gfCNCPoint3[27581] = {X 474.4193, Y 40.3571, Z -4.6667, A 0.000, B 0.000, C 0.000 }
gfCNCPoint3[27582] = {X 478.5504, Y 32.2710, Z -4.6667, A 0.000, B 0.000, C 0.000 }
gfCNCPoint3[27583] = {X 477.2666, Y 31.4237, Z -4.6667, A 0.000, B 0.000, C 0.000 }
gfCNCPoint3[27584] = {X 476.1107, Y 30.4089, Z -4.6667, A 0.000, B 0.000, C 0.000 }
gfCNCPoint3[27585] = {X 475.1043, Y 29.2457, Z -4.6667, A 0.000, B 0.000, C 0.000 }
gfCNCPoint3[27586] = {X 474.2663, Y 27.9559, Z -4.6667, A 0.000, B 0.000, C 0.000 }
gfCNCPoint3[27587] = {X 473.6124, Y 26.5637, Z -4.6667, A 0.000, B 0.000, C 0.000 }
gfCNCPoint3[27588] = {X 473.1548, Y 25.0952, Z -4.6667, A 0.000, B 0.000, C 0.000 }
gfCNCPoint3[27589] = {X 472.8451, Y 23.4362, Z -4.6667, A 0.000, B 0.000, C 0.000 }
gfCNCPoint3[27590] = {X 472.7065, Y 21.7542, Z -4.6667, A 0.000, B 0.000, C 0.000 }
gfCNCPoint3[27591] = {X 472.7407, Y 20.0669, Z -4.6667, A 0.000, B 0.000, C 0.000 }
gfCNCPoint3[27592] = {X 472.9473, Y 18.3920, Z -4.6667, A 0.000, B 0.000, C 0.000 }
gfCNCPoint3[27593] = {X 473.3241, Y 16.7469, Z -4.6667, A 0.000, B 0.000, C 0.000 }
gfCNCPoint3[27594] = {X 473.8558, Y 15.2628, Z -4.6667, A 0.000, B 0.000, C 0.000 }
gfCNCPoint3[27595] = {X 474.5840, Y 13.8645, Z -4.6667, A 0.000, B 0.000, C 0.000 }
gfCNCPoint3[27596] = {X 475.4953, Y 12.5780, Z -4.6667, A 0.000, B 0.000, C 0.000 }
gfCNCPoint3[27597] = {X 476.5726, Y 11.4271, Z -4.6667, A 0.000, B 0.000, C 0.000 }
gfCNCPoint3[27598] = {X 477.7962, Y 10.4330, Z -4.6667, A 0.000, B 0.000, C 0.000 }
gfCNCPoint3[27599] = {X 479.1434, Y 9.6141, Z -4.6667, A 0.000, B 0.000, C 0.000 }
gfCNCPoint3[27600] = {X 480.5892, Y 8.9856, Z -4.6667, A 0.000, B 0.000, C 0.000 }
gfCNCPoint3[27601] = {X 482.1069, Y 8.5592, Z -4.6667, A 0.000, B 0.000, C 0.000 }
gfCNCPoint3[27602] = {X 484.1811, Y 8.2359, Z -4.6667, A 0.000, B 0.000, C 0.000 }
gfCNCPoint3[27603] = {X 486.2773, Y 8.1227, Z -4.6667, A 0.000, B 0.000, C 0.000 }
gfCNCPoint3[27604] = {X 486.9700, Y 8.1106, Z -4.6667, A 0.000, B 0.000, C 0.000 }
gfCNCPoint3[27605] = {X 492.3835, Y 8.1106, Z -4.6667, A 0.000, B 0.000, C 0.000 }
gfCNCPoint3[27606] = {X 492.3835, Y 4.1106, Z -4.6667, A 0.000, B 0.000, C 0.000 }
gfCNCPoint3[27607] = {X 492.3835, Y 8.1906, Z -4.6667, A 0.000, B 0.000, C 0.000 }
gfCNCPoint3[27608] = {X 502.2053, Y 8.1906, Z -4.6667, A 0.000, B 0.000, C 0.000 }
gfCNCPoint3[27609] = {X 502.7369, Y 8.1947, Z -4.6667, A 0.000, B 0.000, C 0.000 }
gfCNCPoint3[27610] = {X 503.6180, Y 8.3005, Z -4.6667, A 0.000, B 0.000, C 0.000 }
gfCNCPoint3[27611] = {X 504.4538, Y 8.5987, Z -4.6667, A 0.000, B 0.000, C 0.000 }
gfCNCPoint3[27612] = {X 505.2029, Y 9.0746, Z -4.6667, A 0.000, B 0.000, C 0.000 }
gfCNCPoint3[27613] = {X 505.8279, Y 9.7045, Z -4.6667, A 0.000, B 0.000, C 0.000 }
gfCNCPoint3[27614] = {X 506.2979, Y 10.4573, Z -4.6667, A 0.000, B 0.000, C 0.000 }
gfCNCPoint3[27615] = {X 506.5896, Y 11.2954, Z -4.6667, A 0.000, B 0.000, C 0.000 }
gfCNCPoint3[27616] = {X 506.6885, Y 12.1773, Z -4.6667, A 0.000, B 0.000, C 0.000 }
gfCNCPoint3[27617] = {X 506.6883, Y 13.0192, Z -4.6667, A 0.000, B 0.000, C 0.000 }
gfCNCPoint3[27618] = {X 506.5797, Y 13.9048, Z -4.6667, A 0.000, B 0.000, C 0.000 }
gfCNCPoint3[27619] = {X 506.2774, Y 14.7443, Z -4.6667, A 0.000, B 0.000, C 0.000 }
gfCNCPoint3[27620] = {X 505.7966, Y 15.4959, Z -4.6667, A 0.000, B 0.000, C 0.000 }
gfCNCPoint3[27621] = {X 505.1612, Y 16.1222, Z -4.6667, A 0.000, B 0.000, C 0.000 }
gfCNCPoint3[27622] = {X 505.1611, Y 41.0655, Z -4.6667, A 0.000, B 0.000, C 0.000 }
gfCNCPoint3[27623] = {X 505.3000, Y 41.1789, Z -4.6667, A 0.000, B 0.000, C 0.000 }
gfCNCPoint3[27624] = {X 505.8859, Y 41.8054, Z -4.6667, A 0.000, B 0.000, C 0.000 }
gfCNCPoint3[27625] = {X 506.3249, Y 42.5424, Z -4.6667, A 0.000, B 0.000, C 0.000 }
gfCNCPoint3[27626] = {X 506.5965, Y 43.3560, Z -4.6667, A 0.000, B 0.000, C 0.000 }
gfCNCPoint3[27627] = {X 506.6885, Y 44.2089, Z -4.6667, A 0.000, B 0.000, C 0.000 }
gfCNCPoint3[27628] = {X 506.6885, Y 45.0000, Z -4.6667, A 0.000, B 0.000, C 0.000 }
gfCNCPoint3[27629] = {X 506.5882, Y 45.8901, Z -4.6667, A 0.000, B 0.000, C 0.000 }
gfCNCPoint3[27630] = {X 506.2924, Y 46.7355, Z -4.6667, A 0.000, B 0.000, C 0.000 }
gfCNCPoint3[27631] = {X 505.8158, Y 47.4940, Z -4.6667, A 0.000, B 0.000, C 0.000 }
gfCNCPoint3[27632] = {X 505.1825, Y 48.1273, Z -4.6667, A 0.000, B 0.000, C 0.000 }
gfCNCPoint3[27633] = {X 504.4240, Y 48.6039, Z -4.6667, A 0.000, B 0.000, C 0.000 }
gfCNCPoint3[27634] = {X 503.5786, Y 48.8997, Z -4.6667, A 0.000, B 0.000, C 0.000 }
gfCNCPoint3[27635] = {X 502.6885, Y 49.0000, Z -4.6667, A 0.000, B 0.000, C 0.000 }
gfCNCPoint3[27636] = {X 496.2450, Y 49.0000, Z -4.6667, A 0.000, B 0.000, C 0.000 }
gfCNCPoint3[27637] = {X 495.3549, Y 48.8997, Z -4.6667, A 0.000, B 0.000, C 0.000 }
gfCNCPoint3[27638] = {X 494.5095, Y 48.6039, Z -4.6667, A 0.000, B 0.000, C 0.000 }
gfCNCPoint3[27639] = {X 493.7511, Y 48.1273, Z -4.6667, A 0.000, B 0.000, C 0.000 }
gfCNCPoint3[27640] = {X 493.1177, Y 47.4939, Z -4.6667, A 0.000, B 0.000, C 0.000 }
gfCNCPoint3[27641] = {X 492.6411, Y 46.7355, Z -4.6667, A 0.000, B 0.000, C 0.000 }
gfCNCPoint3[27642] = {X 492.3453, Y 45.8901, Z -4.6667, A 0.000, B 0.000, C 0.000 }
gfCNCPoint3[27643] = {X 492.2450, Y 45.0000, Z -4.6667, A 0.000, B 0.000, C 0.000 }
gfCNCPoint3[27644] = {X 492.2454, Y 44.1538, Z -4.6667, A 0.000, B 0.000, C 0.000 }
gfCNCPoint3[27645] = {X 492.3560, Y 43.2730, Z -4.6667, A 0.000, B 0.000, C 0.000 }
gfCNCPoint3[27646] = {X 492.6582, Y 42.4382, Z -4.6667, A 0.000, B 0.000, C 0.000 }
gfCNCPoint3[27647] = {X 493.1371, Y 41.6907, Z -4.6667, A 0.000, B 0.000, C 0.000 }
gfCNCPoint3[27648] = {X 493.7690, Y 41.0672, Z -4.6667, A 0.000, B 0.000, C 0.000 }
gfCNCPoint3[27649] = {X 493.7690, Y 34.1538, Z -4.6667, A 0.000, B 0.000, C 0.000 }
gfCNCPoint3[27650] = {X 490.7733, Y 34.1538, Z -4.6667, A 0.000, B 0.000, C 0.000 }
gfCNCPoint3[27651] = {X 490.5302, Y 34.1516, Z -4.6667, A 0.000, B 0.000, C 0.000 }
gfCNCPoint3[27652] = {X 486.0908, Y 42.7966, Z -4.6667, A 0.000, B 0.000, C 0.000 }
gfCNCPoint3[27653] = {X 486.1474, Y 42.9488, Z -4.6667, A 0.000, B 0.000, C 0.000 }
gfCNCPoint3[27654] = {X 486.2998, Y 43.5707, Z -4.6667, A 0.000, B 0.000, C 0.000 }
gfCNCPoint3[27655] = {X 486.3510, Y 44.2089, Z -4.6667, A 0.000, B 0.000, C 0.000 }
gfCNCPoint3[27656] = {X 486.3510, Y 45.0000, Z -4.6667, A 0.000, B 0.000, C 0.000 }
gfCNCPoint3[27657] = {X 486.2507, Y 45.8901, Z -4.6667, A 0.000, B 0.000, C 0.000 }
gfCNCPoint3[27658] = {X 485.9549, Y 46.7355, Z -4.6667, A 0.000, B 0.000, C 0.000 }
gfCNCPoint3[27659] = {X 485.4783, Y 47.4940, Z -4.6667, A 0.000, B 0.000, C 0.000 }
gfCNCPoint3[27660] = {X 484.8450, Y 48.1273, Z -4.6667, A 0.000, B 0.000, C 0.000 }
gfCNCPoint3[27661] = {X 484.0866, Y 48.6039, Z -4.6667, A 0.000, B 0.000, C 0.000 }
gfCNCPoint3[27662] = {X 483.2411, Y 48.8997, Z -4.6667, A 0.000, B 0.000, C 0.000 }
gfCNCPoint3[27663] = {X 482.3510, Y 49.0000, Z -4.6667, A 0.000, B 0.000, C 0.000 }
gfCNCPoint3[27664] = {X 475.7650, Y 49.0000, Z -4.6667, A 0.000, B 0.000, C 0.000 }
gfCNCPoint3[27665] = {X 474.8749, Y 48.8997, Z -4.6667, A 0.000, B 0.000, C 0.000 }
gfCNCPoint3[27666] = {X 474.0294, Y 48.6039, Z -4.6667, A 0.000, B 0.000, C 0.000 }
gfCNCPoint3[27667] = {X 473.2710, Y 48.1273, Z -4.6667, A 0.000, B 0.000, C 0.000 }
gfCNCPoint3[27668] = {X 472.6376, Y 47.4940, Z -4.6667, A 0.000, B 0.000, C 0.000 }
gfCNCPoint3[27669] = {X 472.1611, Y 46.7355, Z -4.6667, A 0.000, B 0.000, C 0.000 }
gfCNCPoint3[27670] = {X 471.8652, Y 45.8901, Z -4.6667, A 0.000, B 0.000, C 0.000 }
gfCNCPoint3[27671] = {X 471.7650, Y 45.0000, Z -4.6667, A 0.000, B 0.000, C 0.000 }
gfCNCPoint3[27672] = {X 471.7653, Y 44.1538, Z -4.6667, A 0.000, B 0.000, C 0.000 }
gfCNCPoint3[27673] = {X 471.8601, Y 43.3414, Z -4.6667, A 0.000, B 0.000, C 0.000 }
gfCNCPoint3[27674] = {X 472.1182, Y 42.5654, Z -4.6667, A 0.000, B 0.000, C 0.000 }
gfCNCPoint3[27675] = {X 472.5286, Y 41.8580, Z -4.6667, A 0.000, B 0.000, C 0.000 }
gfCNCPoint3[27676] = {X 473.0744, Y 41.2489, Z -4.6667, A 0.000, B 0.000, C 0.000 }
gfCNCPoint3[27677] = {X 473.7327, Y 40.7635, Z -4.6667, A 0.000, B 0.000, C 0.000 }
gfCNCPoint3[27678] = {X 474.4759, Y 40.4222, Z -4.6667, A 0.000, B 0.000, C 0.000 }
gfCNCPoint3[27679] = {X 478.6566, Y 32.2388, Z -4.6667, A 0.000, B 0.000, C 0.000 }
gfCNCPoint3[27680] = {X 477.3660, Y 31.3987, Z -4.6667, A 0.000, B 0.000, C 0.000 }
gfCNCPoint3[27681] = {X 476.2035, Y 30.3887, Z -4.6667, A 0.000, B 0.000, C 0.000 }
gfCNCPoint3[27682] = {X 475.1913, Y 29.2282, Z -4.6667, A 0.000, B 0.000, C 0.000 }
gfCNCPoint3[27683] = {X 474.3486, Y 27.9393, Z -4.6667, A 0.000, B 0.000, C 0.000 }
gfCNCPoint3[27684] = {X 473.6915, Y 26.5465, Z -4.6667, A 0.000, B 0.000, C 0.000 }
gfCNCPoint3[27685] = {X 473.2327, Y 25.0766, Z -4.6667, A 0.000, B 0.000, C 0.000 }
gfCNCPoint3[27686] = {X 472.9244, Y 23.4256, Z -4.6667, A 0.000, B 0.000, C 0.000 }
gfCNCPoint3[27687] = {X 472.7865, Y 21.7518, Z -4.6667, A 0.000, B 0.000, C 0.000 }
gfCNCPoint3[27688] = {X 472.8205, Y 20.0727, Z -4.6667, A 0.000, B 0.000, C 0.000 }
gfCNCPoint3[27689] = {X 473.0261, Y 18.4058, Z -4.6667, A 0.000, B 0.000, C 0.000 }
gfCNCPoint3[27690] = {X 473.4010, Y 16.7687, Z -4.6667, A 0.000, B 0.000, C 0.000 }
gfCNCPoint3[27691] = {X 473.9291, Y 15.2948, Z -4.6667, A 0.000, B 0.000, C 0.000 }
gfCNCPoint3[27692] = {X 474.6523, Y 13.9062, Z -4.6667, A 0.000, B 0.000, C 0.000 }
gfCNCPoint3[27693] = {X 475.5572, Y 12.6286, Z -4.6667, A 0.000, B 0.000, C 0.000 }
gfCNCPoint3[27694] = {X 476.6272, Y 11.4856, Z -4.6667, A 0.000, B 0.000, C 0.000 }
gfCNCPoint3[27695] = {X 477.8423, Y 10.4984, Z -4.6667, A 0.000, B 0.000, C 0.000 }
gfCNCPoint3[27696] = {X 479.1802, Y 9.6851, Z -4.6667, A 0.000, B 0.000, C 0.000 }
gfCNCPoint3[27697] = {X 480.6160, Y 9.0610, Z -4.6667, A 0.000, B 0.000, C 0.000 }
gfCNCPoint3[27698] = {X 482.1233, Y 8.6375, Z -4.6667, A 0.000, B 0.000, C 0.000 }
gfCNCPoint3[27699] = {X 484.1898, Y 8.3155, Z -4.6667, A 0.000, B 0.000, C 0.000 }
gfCNCPoint3[27700] = {X 486.2782, Y 8.2027, Z -4.6667, A 0.000, B 0.000, C 0.000 }
gfCNCPoint3[27701] = {X 486.9707, Y 8.1906, Z -4.6667, A 0.000, B 0.000, C 0.000 }
gfCNCPoint3[27702] = {X 492.3835, Y 8.1906, Z -4.6667, A 0.000, B 0.000, C 0.000 }
gfCNCPoint3[27703] = {X 492.3835, Y 4.1106, Z -4.6667, A 0.000, B 0.000, C 0.000 }
gfCNCPoint3[27704] = {X 492.3835, Y 4.1106, Z -1.6667, A 0.000, B 0.000, C 0.000 }
gfCNCPoint3[27705] = {X 492.3835, Y 4.1106, Z 11.0000, A 0.000, B 0.000, C 0.000 }
gfCNCPoint3[27706] = {X 533.9637, Y 3.7903, Z 11.0000, A 0.000, B 0.000, C 0.000 }
gfCNCPoint3[27707] = {X 533.9637, Y 3.7903, Z -1.6667, A 0.000, B 0.000, C 0.000 }
gfCNCPoint3[27708] = {X 533.9637, Y 3.7903, Z -4.6667, A 0.000, B 0.000, C 0.000 }
gfCNCPoint3[27709] = {X 533.9636, Y 7.8703, Z -4.6667, A 0.000, B 0.000, C 0.000 }
gfCNCPoint3[27710] = {X 543.7499, Y 7.8706, Z -4.6667, A 0.000, B 0.000, C 0.000 }
gfCNCPoint3[27711] = {X 544.7301, Y 7.9561, Z -4.6667, A 0.000, B 0.000, C 0.000 }
gfCNCPoint3[27712] = {X 545.6657, Y 8.2610, Z -4.6667, A 0.000, B 0.000, C 0.000 }
gfCNCPoint3[27713] = {X 546.5081, Y 8.7694, Z -4.6667, A 0.000, B 0.000, C 0.000 }
gfCNCPoint3[27714] = {X 547.2138, Y 9.4551, Z -4.6667, A 0.000, B 0.000, C 0.000 }
gfCNCPoint3[27715] = {X 547.7462, Y 10.2825, Z -4.6667, A 0.000, B 0.000, C 0.000 }
gfCNCPoint3[27716] = {X 548.0778, Y 11.2089, Z -4.6667, A 0.000, B 0.000, C 0.000 }
gfCNCPoint3[27717] = {X 548.1914, Y 12.1863, Z -4.6667, A 0.000, B 0.000, C 0.000 }
gfCNCPoint3[27718] = {X 548.1912, Y 13.0225, Z -4.6667, A 0.000, B 0.000, C 0.000 }
gfCNCPoint3[27719] = {X 548.0827, Y 13.9405, Z -4.6667, A 0.000, B 0.000, C 0.000 }
gfCNCPoint3[27720] = {X 547.7815, Y 14.8144, Z -4.6667, A 0.000, B 0.000, C 0.000 }
gfCNCPoint3[27721] = {X 547.3012, Y 15.6043, Z -4.6667, A 0.000, B 0.000, C 0.000 }
gfCNCPoint3[27722] = {X 546.6638, Y 16.2738, Z -4.6667, A 0.000, B 0.000, C 0.000 }
gfCNCPoint3[27723] = {X 546.6640, Y 40.9136, Z -4.6667, A 0.000, B 0.000, C 0.000 }
gfCNCPoint3[27724] = {X 546.6861, Y 40.9316, Z -4.6667, A 0.000, B 0.000, C 0.000 }
gfCNCPoint3[27725] = {X 547.3159, Y 41.6015, Z -4.6667, A 0.000, B 0.000, C 0.000 }
gfCNCPoint3[27726] = {X 547.7897, Y 42.3895, Z -4.6667, A 0.000, B 0.000, C 0.000 }
gfCNCPoint3[27727] = {X 548.0859, Y 43.2599, Z -4.6667, A 0.000, B 0.000, C 0.000 }
gfCNCPoint3[27728] = {X 548.1913, Y 44.1733, Z -4.6667, A 0.000, B 0.000, C 0.000 }
gfCNCPoint3[27729] = {X 548.1914, Y 45.0005, Z -4.6667, A 0.000, B 0.000, C 0.000 }
gfCNCPoint3[27730] = {X 548.0778, Y 45.9779, Z -4.6667, A 0.000, B 0.000, C 0.000 }
gfCNCPoint3[27731] = {X 547.7462, Y 46.9042, Z -4.6667, A 0.000, B 0.000, C 0.000 }
gfCNCPoint3[27732] = {X 547.2138, Y 47.7317, Z -4.6667, A 0.000, B 0.000, C 0.000 }
gfCNCPoint3[27733] = {X 546.5081, Y 48.4173, Z -4.6667, A 0.000, B 0.000, C 0.000 }
gfCNCPoint3[27734] = {X 545.6657, Y 48.9257, Z -4.6667, A 0.000, B 0.000, C 0.000 }
gfCNCPoint3[27735] = {X 544.7301, Y 49.2305, Z -4.6667, A 0.000, B 0.000, C 0.000 }
gfCNCPoint3[27736] = {X 543.7499, Y 49.3159, Z -4.6667, A 0.000, B 0.000, C 0.000 }
gfCNCPoint3[27737] = {X 524.0451, Y 49.3164, Z -4.6667, A 0.000, B 0.000, C 0.000 }
gfCNCPoint3[27738] = {X 523.4986, Y 49.9503, Z -4.6667, A 0.000, B 0.000, C 0.000 }
gfCNCPoint3[27739] = {X 522.8436, Y 50.4714, Z -4.6667, A 0.000, B 0.000, C 0.000 }
gfCNCPoint3[27740] = {X 522.1030, Y 50.8615, Z -4.6667, A 0.000, B 0.000, C 0.000 }
gfCNCPoint3[27741] = {X 521.3028, Y 51.1069, Z -4.6667, A 0.000, B 0.000, C 0.000 }
gfCNCPoint3[27742] = {X 520.4709, Y 51.1991, Z -4.6667, A 0.000, B 0.000, C 0.000 }
gfCNCPoint3[27743] = {X 519.7998, Y 51.1991, Z -4.6667, A 0.000, B 0.000, C 0.000 }
gfCNCPoint3[27744] = {X 518.8385, Y 51.0908, Z -4.6667, A 0.000, B 0.000, C 0.000 }
gfCNCPoint3[27745] = {X 517.9254, Y 50.7713, Z -4.6667, A 0.000, B 0.000, C 0.000 }
gfCNCPoint3[27746] = {X 517.1063, Y 50.2566, Z -4.6667, A 0.000, B 0.000, C 0.000 }
gfCNCPoint3[27747] = {X 516.4223, Y 49.5726, Z -4.6667, A 0.000, B 0.000, C 0.000 }
gfCNCPoint3[27748] = {X 515.9076, Y 48.7535, Z -4.6667, A 0.000, B 0.000, C 0.000 }
gfCNCPoint3[27749] = {X 515.5881, Y 47.8404, Z -4.6667, A 0.000, B 0.000, C 0.000 }
gfCNCPoint3[27750] = {X 515.4798, Y 46.8791, Z -4.6667, A 0.000, B 0.000, C 0.000 }
gfCNCPoint3[27751] = {X 515.4798, Y 39.9011, Z -4.6667, A 0.000, B 0.000, C 0.000 }
gfCNCPoint3[27752] = {X 515.5869, Y 38.9451, Z -4.6667, A 0.000, B 0.000, C 0.000 }
gfCNCPoint3[27753] = {X 515.9029, Y 38.0365, Z -4.6667, A 0.000, B 0.000, C 0.000 }
gfCNCPoint3[27754] = {X 516.4121, Y 37.2204, Z -4.6667, A 0.000, B 0.000, C 0.000 }
gfCNCPoint3[27755] = {X 517.0893, Y 36.5372, Z -4.6667, A 0.000, B 0.000, C 0.000 }
gfCNCPoint3[27756] = {X 517.9010, Y 36.0208, Z -4.6667, A 0.000, B 0.000, C 0.000 }
gfCNCPoint3[27757] = {X 518.8067, Y 35.6968, Z -4.6667, A 0.000, B 0.000, C 0.000 }
gfCNCPoint3[27758] = {X 519.7617, Y 35.5813, Z -4.6667, A 0.000, B 0.000, C 0.000 }
gfCNCPoint3[27759] = {X 520.5269, Y 35.5815, Z -4.6667, A 0.000, B 0.000, C 0.000 }
gfCNCPoint3[27760] = {X 521.3533, Y 35.6728, Z -4.6667, A 0.000, B 0.000, C 0.000 }
gfCNCPoint3[27761] = {X 522.1470, Y 35.9207, Z -4.6667, A 0.000, B 0.000, C 0.000 }
gfCNCPoint3[27762] = {X 522.8785, Y 36.3160, Z -4.6667, A 0.000, B 0.000, C 0.000 }
gfCNCPoint3[27763] = {X 523.5207, Y 36.8442, Z -4.6667, A 0.000, B 0.000, C 0.000 }
gfCNCPoint3[27764] = {X 524.0498, Y 37.4856, Z -4.6667, A 0.000, B 0.000, C 0.000 }
gfCNCPoint3[27765] = {X 534.6319, Y 37.4861, Z -4.6667, A 0.000, B 0.000, C 0.000 }
gfCNCPoint3[27766] = {X 534.6319, Y 33.9655, Z -4.6667, A 0.000, B 0.000, C 0.000 }
gfCNCPoint3[27767] = {X 530.1088, Y 33.9668, Z -4.6667, A 0.000, B 0.000, C 0.000 }
gfCNCPoint3[27768] = {X 529.5766, Y 34.6107, Z -4.6667, A 0.000, B 0.000, C 0.000 }
gfCNCPoint3[27769] = {X 528.9304, Y 35.1401, Z -4.6667, A 0.000, B 0.000, C 0.000 }
gfCNCPoint3[27770] = {X 528.1944, Y 35.5353, Z -4.6667, A 0.000, B 0.000, C 0.000 }
gfCNCPoint3[27771] = {X 527.3962, Y 35.7814, Z -4.6667, A 0.000, B 0.000, C 0.000 }
gfCNCPoint3[27772] = {X 526.5655, Y 35.8693, Z -4.6667, A 0.000, B 0.000, C 0.000 }
gfCNCPoint3[27773] = {X 525.8868, Y 35.8694, Z -4.6667, A 0.000, B 0.000, C 0.000 }
gfCNCPoint3[27774] = {X 524.9255, Y 35.7611, Z -4.6667, A 0.000, B 0.000, C 0.000 }
gfCNCPoint3[27775] = {X 524.0124, Y 35.4416, Z -4.6667, A 0.000, B 0.000, C 0.000 }
gfCNCPoint3[27776] = {X 523.1933, Y 34.9270, Z -4.6667, A 0.000, B 0.000, C 0.000 }
gfCNCPoint3[27777] = {X 522.5092, Y 34.2429, Z -4.6667, A 0.000, B 0.000, C 0.000 }
gfCNCPoint3[27778] = {X 521.9946, Y 33.4238, Z -4.6667, A 0.000, B 0.000, C 0.000 }
gfCNCPoint3[27779] = {X 521.6751, Y 32.5107, Z -4.6667, A 0.000, B 0.000, C 0.000 }
gfCNCPoint3[27780] = {X 521.5668, Y 31.5495, Z -4.6667, A 0.000, B 0.000, C 0.000 }
gfCNCPoint3[27781] = {X 521.5668, Y 24.5714, Z -4.6667, A 0.000, B 0.000, C 0.000 }
gfCNCPoint3[27782] = {X 521.6739, Y 23.6153, Z -4.6667, A 0.000, B 0.000, C 0.000 }
gfCNCPoint3[27783] = {X 521.9900, Y 22.7066, Z -4.6667, A 0.000, B 0.000, C 0.000 }
gfCNCPoint3[27784] = {X 522.4994, Y 21.8904, Z -4.6667, A 0.000, B 0.000, C 0.000 }
gfCNCPoint3[27785] = {X 523.1768, Y 21.2071, Z -4.6667, A 0.000, B 0.000, C 0.000 }
gfCNCPoint3[27786] = {X 523.9886, Y 20.6908, Z -4.6667, A 0.000, B 0.000, C 0.000 }
gfCNCPoint3[27787] = {X 524.8946, Y 20.3669, Z -4.6667, A 0.000, B 0.000, C 0.000 }
gfCNCPoint3[27788] = {X 525.8498, Y 20.2516, Z -4.6667, A 0.000, B 0.000, C 0.000 }
gfCNCPoint3[27789] = {X 526.5695, Y 20.2516, Z -4.6667, A 0.000, B 0.000, C 0.000 }
gfCNCPoint3[27790] = {X 527.3945, Y 20.3391, Z -4.6667, A 0.000, B 0.000, C 0.000 }
gfCNCPoint3[27791] = {X 528.1876, Y 20.5828, Z -4.6667, A 0.000, B 0.000, C 0.000 }
gfCNCPoint3[27792] = {X 528.9195, Y 20.9735, Z -4.6667, A 0.000, B 0.000, C 0.000 }
gfCNCPoint3[27793] = {X 529.5632, Y 21.4970, Z -4.6667, A 0.000, B 0.000, C 0.000 }
gfCNCPoint3[27794] = {X 530.0950, Y 22.1338, Z -4.6667, A 0.000, B 0.000, C 0.000 }
gfCNCPoint3[27795] = {X 534.6319, Y 22.1341, Z -4.6667, A 0.000, B 0.000, C 0.000 }
gfCNCPoint3[27796] = {X 534.6319, Y 19.7019, Z -4.6667, A 0.000, B 0.000, C 0.000 }
gfCNCPoint3[27797] = {X 524.1921, Y 19.7016, Z -4.6667, A 0.000, B 0.000, C 0.000 }
gfCNCPoint3[27798] = {X 523.6597, Y 20.3462, Z -4.6667, A 0.000, B 0.000, C 0.000 }
gfCNCPoint3[27799] = {X 523.0130, Y 20.8762, Z -4.6667, A 0.000, B 0.000, C 0.000 }
gfCNCPoint3[27800] = {X 522.2764, Y 21.2717, Z -4.6667, A 0.000, B 0.000, C 0.000 }
gfCNCPoint3[27801] = {X 521.4774, Y 21.5179, Z -4.6667, A 0.000, B 0.000, C 0.000 }
gfCNCPoint3[27802] = {X 520.6460, Y 21.6056, Z -4.6667, A 0.000, B 0.000, C 0.000 }
gfCNCPoint3[27803] = {X 519.9691, Y 21.6057, Z -4.6667, A 0.000, B 0.000, C 0.000 }
gfCNCPoint3[27804] = {X 519.0078, Y 21.4974, Z -4.6667, A 0.000, B 0.000, C 0.000 }
gfCNCPoint3[27805] = {X 518.0947, Y 21.1779, Z -4.6667, A 0.000, B 0.000, C 0.000 }
gfCNCPoint3[27806] = {X 517.2756, Y 20.6632, Z -4.6667, A 0.000, B 0.000, C 0.000 }
gfCNCPoint3[27807] = {X 516.5916, Y 19.9792, Z -4.6667, A 0.000, B 0.000, C 0.000 }
gfCNCPoint3[27808] = {X 516.0769, Y 19.1601, Z -4.6667, A 0.000, B 0.000, C 0.000 }
gfCNCPoint3[27809] = {X 515.7574, Y 18.2470, Z -4.6667, A 0.000, B 0.000, C 0.000 }
gfCNCPoint3[27810] = {X 515.6491, Y 17.2857, Z -4.6667, A 0.000, B 0.000, C 0.000 }
gfCNCPoint3[27811] = {X 515.6491, Y 10.3077, Z -4.6667, A 0.000, B 0.000, C 0.000 }
gfCNCPoint3[27812] = {X 515.7562, Y 9.3519, Z -4.6667, A 0.000, B 0.000, C 0.000 }
gfCNCPoint3[27813] = {X 516.0720, Y 8.4435, Z -4.6667, A 0.000, B 0.000, C 0.000 }
gfCNCPoint3[27814] = {X 516.5811, Y 7.6275, Z -4.6667, A 0.000, B 0.000, C 0.000 }
gfCNCPoint3[27815] = {X 517.2580, Y 6.9443, Z -4.6667, A 0.000, B 0.000, C 0.000 }
gfCNCPoint3[27816] = {X 518.0693, Y 6.4278, Z -4.6667, A 0.000, B 0.000, C 0.000 }
gfCNCPoint3[27817] = {X 518.9748, Y 6.1037, Z -4.6667, A 0.000, B 0.000, C 0.000 }
gfCNCPoint3[27818] = {X 519.9296, Y 5.9879, Z -4.6667, A 0.000, B 0.000, C 0.000 }
gfCNCPoint3[27819] = {X 520.6502, Y 5.9879, Z -4.6667, A 0.000, B 0.000, C 0.000 }
gfCNCPoint3[27820] = {X 521.4756, Y 6.0751, Z -4.6667, A 0.000, B 0.000, C 0.000 }
gfCNCPoint3[27821] = {X 522.2691, Y 6.3187, Z -4.6667, A 0.000, B 0.000, C 0.000 }
gfCNCPoint3[27822] = {X 523.0013, Y 6.7094, Z -4.6667, A 0.000, B 0.000, C 0.000 }
gfCNCPoint3[27823] = {X 523.6454, Y 7.2330, Z -4.6667, A 0.000, B 0.000, C 0.000 }
gfCNCPoint3[27824] = {X 524.1774, Y 7.8701, Z -4.6667, A 0.000, B 0.000, C 0.000 }
gfCNCPoint3[27825] = {X 533.9636, Y 7.8703, Z -4.6667, A 0.000, B 0.000, C 0.000 }
gfCNCPoint3[27826] = {X 533.9637, Y 3.8703, Z -4.6667, A 0.000, B 0.000, C 0.000 }
gfCNCPoint3[27827] = {X 533.9636, Y 7.9503, Z -4.6667, A 0.000, B 0.000, C 0.000 }
gfCNCPoint3[27828] = {X 543.7510, Y 7.9506, Z -4.6667, A 0.000, B 0.000, C 0.000 }
gfCNCPoint3[27829] = {X 544.7133, Y 8.0343, Z -4.6667, A 0.000, B 0.000, C 0.000 }
gfCNCPoint3[27830] = {X 545.6317, Y 8.3334, Z -4.6667, A 0.000, B 0.000, C 0.000 }
gfCNCPoint3[27831] = {X 546.4587, Y 8.8324, Z -4.6667, A 0.000, B 0.000, C 0.000 }
gfCNCPoint3[27832] = {X 547.1515, Y 9.5054, Z -4.6667, A 0.000, B 0.000, C 0.000 }
gfCNCPoint3[27833] = {X 547.6743, Y 10.3176, Z -4.6667, A 0.000, B 0.000, C 0.000 }
gfCNCPoint3[27834] = {X 547.9999, Y 11.2270, Z -4.6667, A 0.000, B 0.000, C 0.000 }
gfCNCPoint3[27835] = {X 548.1114, Y 12.1864, Z -4.6667, A 0.000, B 0.000, C 0.000 }
gfCNCPoint3[27836] = {X 548.1112, Y 13.0217, Z -4.6667, A 0.000, B 0.000, C 0.000 }
gfCNCPoint3[27837] = {X 548.0027, Y 13.9317, Z -4.6667, A 0.000, B 0.000, C 0.000 }
gfCNCPoint3[27838] = {X 547.7012, Y 14.7971, Z -4.6667, A 0.000, B 0.000, C 0.000 }
gfCNCPoint3[27839] = {X 547.2207, Y 15.5776, Z -4.6667, A 0.000, B 0.000, C 0.000 }
gfCNCPoint3[27840] = {X 546.5838, Y 16.2365, Z -4.6667, A 0.000, B 0.000, C 0.000 }
gfCNCPoint3[27841] = {X 546.5840, Y 40.9517, Z -4.6667, A 0.000, B 0.000, C 0.000 }
gfCNCPoint3[27842] = {X 546.6348, Y 40.9930, Z -4.6667, A 0.000, B 0.000, C 0.000 }
gfCNCPoint3[27843] = {X 547.2526, Y 41.6504, Z -4.6667, A 0.000, B 0.000, C 0.000 }
gfCNCPoint3[27844] = {X 547.7173, Y 42.4237, Z -4.6667, A 0.000, B 0.000, C 0.000 }
gfCNCPoint3[27845] = {X 548.0079, Y 43.2777, Z -4.6667, A 0.000, B 0.000, C 0.000 }
gfCNCPoint3[27846] = {X 548.1113, Y 44.1740, Z -4.6667, A 0.000, B 0.000, C 0.000 }
gfCNCPoint3[27847] = {X 548.1114, Y 45.0004, Z -4.6667, A 0.000, B 0.000, C 0.000 }
gfCNCPoint3[27848] = {X 547.9999, Y 45.9598, Z -4.6667, A 0.000, B 0.000, C 0.000 }
gfCNCPoint3[27849] = {X 547.6743, Y 46.8692, Z -4.6667, A 0.000, B 0.000, C 0.000 }
gfCNCPoint3[27850] = {X 547.1516, Y 47.6814, Z -4.6667, A 0.000, B 0.000, C 0.000 }
gfCNCPoint3[27851] = {X 546.4587, Y 48.3544, Z -4.6667, A 0.000, B 0.000, C 0.000 }
gfCNCPoint3[27852] = {X 545.6317, Y 48.8533, Z -4.6667, A 0.000, B 0.000, C 0.000 }
gfCNCPoint3[27853] = {X 544.7133, Y 49.1523, Z -4.6667, A 0.000, B 0.000, C 0.000 }
gfCNCPoint3[27854] = {X 543.7510, Y 49.2359, Z -4.6667, A 0.000, B 0.000, C 0.000 }
gfCNCPoint3[27855] = {X 524.0036, Y 49.2364, Z -4.6667, A 0.000, B 0.000, C 0.000 }
gfCNCPoint3[27856] = {X 523.4669, Y 49.8696, Z -4.6667, A 0.000, B 0.000, C 0.000 }
gfCNCPoint3[27857] = {X 522.8207, Y 50.3907, Z -4.6667, A 0.000, B 0.000, C 0.000 }
gfCNCPoint3[27858] = {X 522.0881, Y 50.7811, Z -4.6667, A 0.000, B 0.000, C 0.000 }
gfCNCPoint3[27859] = {X 521.2951, Y 51.0268, Z -4.6667, A 0.000, B 0.000, C 0.000 }
gfCNCPoint3[27860] = {X 520.4702, Y 51.1191, Z -4.6667, A 0.000, B 0.000, C 0.000 }
gfCNCPoint3[27861] = {X 519.7998, Y 51.1191, Z -4.6667, A 0.000, B 0.000, C 0.000 }
gfCNCPoint3[27862] = {X 518.8563, Y 51.0128, Z -4.6667, A 0.000, B 0.000, C 0.000 }
gfCNCPoint3[27863] = {X 517.9601, Y 50.6992, Z -4.6667, A 0.000, B 0.000, C 0.000 }
gfCNCPoint3[27864] = {X 517.1562, Y 50.1941, Z -4.6667, A 0.000, B 0.000, C 0.000 }
gfCNCPoint3[27865] = {X 516.4848, Y 49.5227, Z -4.6667, A 0.000, B 0.000, C 0.000 }
gfCNCPoint3[27866] = {X 515.9797, Y 48.7188, Z -4.6667, A 0.000, B 0.000, C 0.000 }
gfCNCPoint3[27867] = {X 515.6661, Y 47.8226, Z -4.6667, A 0.000, B 0.000, C 0.000 }
gfCNCPoint3[27868] = {X 515.5598, Y 46.8791, Z -4.6667, A 0.000, B 0.000, C 0.000 }
gfCNCPoint3[27869] = {X 515.5598, Y 39.9011, Z -4.6667, A 0.000, B 0.000, C 0.000 }
gfCNCPoint3[27870] = {X 515.6649, Y 38.9628, Z -4.6667, A 0.000, B 0.000, C 0.000 }
gfCNCPoint3[27871] = {X 515.9751, Y 38.0710, Z -4.6667, A 0.000, B 0.000, C 0.000 }
gfCNCPoint3[27872] = {X 516.4749, Y 37.2700, Z -4.6667, A 0.000, B 0.000, C 0.000 }
gfCNCPoint3[27873] = {X 517.1395, Y 36.5995, Z -4.6667, A 0.000, B 0.000, C 0.000 }
gfCNCPoint3[27874] = {X 517.9361, Y 36.0926, Z -4.6667, A 0.000, B 0.000, C 0.000 }
gfCNCPoint3[27875] = {X 518.8251, Y 35.7746, Z -4.6667, A 0.000, B 0.000, C 0.000 }
gfCNCPoint3[27876] = {X 519.7624, Y 35.6613, Z -4.6667, A 0.000, B 0.000, C 0.000 }
gfCNCPoint3[27877] = {X 520.5258, Y 35.6615, Z -4.6667, A 0.000, B 0.000, C 0.000 }
gfCNCPoint3[27878] = {X 521.3452, Y 35.7528, Z -4.6667, A 0.000, B 0.000, C 0.000 }
gfCNCPoint3[27879] = {X 522.1315, Y 36.0010, Z -4.6667, A 0.000, B 0.000, C 0.000 }
gfCNCPoint3[27880] = {X 522.8549, Y 36.3967, Z -4.6667, A 0.000, B 0.000, C 0.000 }
gfCNCPoint3[27881] = {X 523.4881, Y 36.9249, Z -4.6667, A 0.000, B 0.000, C 0.000 }
gfCNCPoint3[27882] = {X 524.0070, Y 37.5656, Z -4.6667, A 0.000, B 0.000, C 0.000 }
gfCNCPoint3[27883] = {X 534.7119, Y 37.5661, Z -4.6667, A 0.000, B 0.000, C 0.000 }
gfCNCPoint3[27884] = {X 534.7119, Y 33.8855, Z -4.6667, A 0.000, B 0.000, C 0.000 }
gfCNCPoint3[27885] = {X 530.0657, Y 33.8851, Z -4.6667, A 0.000, B 0.000, C 0.000 }
gfCNCPoint3[27886] = {X 530.0418, Y 33.9231, Z -4.6667, A 0.000, B 0.000, C 0.000 }
gfCNCPoint3[27887] = {X 529.5194, Y 34.5547, Z -4.6667, A 0.000, B 0.000, C 0.000 }
gfCNCPoint3[27888] = {X 528.8853, Y 35.0740, Z -4.6667, A 0.000, B 0.000, C 0.000 }
gfCNCPoint3[27889] = {X 528.1631, Y 35.4617, Z -4.6667, A 0.000, B 0.000, C 0.000 }
gfCNCPoint3[27890] = {X 527.3799, Y 35.7031, Z -4.6667, A 0.000, B 0.000, C 0.000 }
gfCNCPoint3[27891] = {X 526.5648, Y 35.7893, Z -4.6667, A 0.000, B 0.000, C 0.000 }
gfCNCPoint3[27892] = {X 525.8868, Y 35.7894, Z -4.6667, A 0.000, B 0.000, C 0.000 }
gfCNCPoint3[27893] = {X 524.9433, Y 35.6831, Z -4.6667, A 0.000, B 0.000, C 0.000 }
gfCNCPoint3[27894] = {X 524.0471, Y 35.3696, Z -4.6667, A 0.000, B 0.000, C 0.000 }
gfCNCPoint3[27895] = {X 523.2432, Y 34.8644, Z -4.6667, A 0.000, B 0.000, C 0.000 }
gfCNCPoint3[27896] = {X 522.5718, Y 34.1930, Z -4.6667, A 0.000, B 0.000, C 0.000 }
gfCNCPoint3[27897] = {X 522.0666, Y 33.3891, Z -4.6667, A 0.000, B 0.000, C 0.000 }
gfCNCPoint3[27898] = {X 521.7531, Y 32.4929, Z -4.6667, A 0.000, B 0.000, C 0.000 }
gfCNCPoint3[27899] = {X 521.6468, Y 31.5495, Z -4.6667, A 0.000, B 0.000, C 0.000 }
gfCNCPoint3[27900] = {X 521.6468, Y 24.5714, Z -4.6667, A 0.000, B 0.000, C 0.000 }
gfCNCPoint3[27901] = {X 521.7519, Y 23.6330, Z -4.6667, A 0.000, B 0.000, C 0.000 }
gfCNCPoint3[27902] = {X 522.0622, Y 22.7411, Z -4.6667, A 0.000, B 0.000, C 0.000 }
gfCNCPoint3[27903] = {X 522.5621, Y 21.9400, Z -4.6667, A 0.000, B 0.000, C 0.000 }
gfCNCPoint3[27904] = {X 523.2270, Y 21.2694, Z -4.6667, A 0.000, B 0.000, C 0.000 }
gfCNCPoint3[27905] = {X 524.0238, Y 20.7626, Z -4.6667, A 0.000, B 0.000, C 0.000 }
gfCNCPoint3[27906] = {X 524.9130, Y 20.4448, Z -4.6667, A 0.000, B 0.000, C 0.000 }
gfCNCPoint3[27907] = {X 525.8505, Y 20.3316, Z -4.6667, A 0.000, B 0.000, C 0.000 }
gfCNCPoint3[27908] = {X 526.5687, Y 20.3316, Z -4.6667, A 0.000, B 0.000, C 0.000 }
gfCNCPoint3[27909] = {X 527.3867, Y 20.4192, Z -4.6667, A 0.000, B 0.000, C 0.000 }
gfCNCPoint3[27910] = {X 528.1724, Y 20.6631, Z -4.6667, A 0.000, B 0.000, C 0.000 }
gfCNCPoint3[27911] = {X 528.8962, Y 21.0542, Z -4.6667, A 0.000, B 0.000, C 0.000 }
gfCNCPoint3[27912] = {X 529.5309, Y 21.5776, Z -4.6667, A 0.000, B 0.000, C 0.000 }
gfCNCPoint3[27913] = {X 530.0525, Y 22.2138, Z -4.6667, A 0.000, B 0.000, C 0.000 }
gfCNCPoint3[27914] = {X 534.7119, Y 22.2141, Z -4.6667, A 0.000, B 0.000, C 0.000 }
gfCNCPoint3[27915] = {X 534.7119, Y 19.6219, Z -4.6667, A 0.000, B 0.000, C 0.000 }
gfCNCPoint3[27916] = {X 524.1491, Y 19.6216, Z -4.6667, A 0.000, B 0.000, C 0.000 }
gfCNCPoint3[27917] = {X 524.1258, Y 19.6568, Z -4.6667, A 0.000, B 0.000, C 0.000 }
gfCNCPoint3[27918] = {X 523.6032, Y 20.2895, Z -4.6667, A 0.000, B 0.000, C 0.000 }
gfCNCPoint3[27919] = {X 522.9686, Y 20.8097, Z -4.6667, A 0.000, B 0.000, C 0.000 }
gfCNCPoint3[27920] = {X 522.2456, Y 21.1979, Z -4.6667, A 0.000, B 0.000, C 0.000 }
gfCNCPoint3[27921] = {X 521.4614, Y 21.4395, Z -4.6667, A 0.000, B 0.000, C 0.000 }
gfCNCPoint3[27922] = {X 520.6453, Y 21.5256, Z -4.6667, A 0.000, B 0.000, C 0.000 }
gfCNCPoint3[27923] = {X 519.9691, Y 21.5257, Z -4.6667, A 0.000, B 0.000, C 0.000 }
gfCNCPoint3[27924] = {X 519.0256, Y 21.4194, Z -4.6667, A 0.000, B 0.000, C 0.000 }
gfCNCPoint3[27925] = {X 518.1294, Y 21.1058, Z -4.6667, A 0.000, B 0.000, C 0.000 }
gfCNCPoint3[27926] = {X 517.3255, Y 20.6007, Z -4.6667, A 0.000, B 0.000, C 0.000 }
gfCNCPoint3[27927] = {X 516.6541, Y 19.9293, Z -4.6667, A 0.000, B 0.000, C 0.000 }
gfCNCPoint3[27928] = {X 516.1490, Y 19.1254, Z -4.6667, A 0.000, B 0.000, C 0.000 }
gfCNCPoint3[27929] = {X 515.8354, Y 18.2292, Z -4.6667, A 0.000, B 0.000, C 0.000 }
gfCNCPoint3[27930] = {X 515.7291, Y 17.2857, Z -4.6667, A 0.000, B 0.000, C 0.000 }
gfCNCPoint3[27931] = {X 515.7291, Y 10.3077, Z -4.6667, A 0.000, B 0.000, C 0.000 }
gfCNCPoint3[27932] = {X 515.8342, Y 9.3696, Z -4.6667, A 0.000, B 0.000, C 0.000 }
gfCNCPoint3[27933] = {X 516.1442, Y 8.4780, Z -4.6667, A 0.000, B 0.000, C 0.000 }
gfCNCPoint3[27934] = {X 516.6438, Y 7.6771, Z -4.6667, A 0.000, B 0.000, C 0.000 }
gfCNCPoint3[27935] = {X 517.3082, Y 7.0066, Z -4.6667, A 0.000, B 0.000, C 0.000 }
gfCNCPoint3[27936] = {X 518.1045, Y 6.4997, Z -4.6667, A 0.000, B 0.000, C 0.000 }
gfCNCPoint3[27937] = {X 518.9932, Y 6.1815, Z -4.6667, A 0.000, B 0.000, C 0.000 }
gfCNCPoint3[27938] = {X 519.9303, Y 6.0679, Z -4.6667, A 0.000, B 0.000, C 0.000 }
gfCNCPoint3[27939] = {X 520.6494, Y 6.0679, Z -4.6667, A 0.000, B 0.000, C 0.000 }
gfCNCPoint3[27940] = {X 521.4678, Y 6.1552, Z -4.6667, A 0.000, B 0.000, C 0.000 }
gfCNCPoint3[27941] = {X 522.2539, Y 6.3990, Z -4.6667, A 0.000, B 0.000, C 0.000 }
gfCNCPoint3[27942] = {X 522.9781, Y 6.7901, Z -4.6667, A 0.000, B 0.000, C 0.000 }
gfCNCPoint3[27943] = {X 523.6130, Y 7.3137, Z -4.6667, A 0.000, B 0.000, C 0.000 }
gfCNCPoint3[27944] = {X 524.1349, Y 7.9501, Z -4.6667, A 0.000, B 0.000, C 0.000 }
gfCNCPoint3[27945] = {X 533.9636, Y 7.9503, Z -4.6667, A 0.000, B 0.000, C 0.000 }
gfCNCPoint3[27946] = {X 533.9637, Y 3.9503, Z -4.6667, A 0.000, B 0.000, C 0.000 }
gfCNCPoint3[27947] = {X 533.9636, Y 8.0303, Z -4.6667, A 0.000, B 0.000, C 0.000 }
gfCNCPoint3[27948] = {X 543.7521, Y 8.0306, Z -4.6667, A 0.000, B 0.000, C 0.000 }
gfCNCPoint3[27949] = {X 544.6964, Y 8.1125, Z -4.6667, A 0.000, B 0.000, C 0.000 }
gfCNCPoint3[27950] = {X 545.5977, Y 8.4058, Z -4.6667, A 0.000, B 0.000, C 0.000 }
gfCNCPoint3[27951] = {X 546.4094, Y 8.8953, Z -4.6667, A 0.000, B 0.000, C 0.000 }
gfCNCPoint3[27952] = {X 547.0893, Y 9.5557, Z -4.6667, A 0.000, B 0.000, C 0.000 }
gfCNCPoint3[27953] = {X 547.6024, Y 10.3527, Z -4.6667, A 0.000, B 0.000, C 0.000 }
gfCNCPoint3[27954] = {X 547.9219, Y 11.2451, Z -4.6667, A 0.000, B 0.000, C 0.000 }
gfCNCPoint3[27955] = {X 548.0314, Y 12.1866, Z -4.6667, A 0.000, B 0.000, C 0.000 }
gfCNCPoint3[27956] = {X 548.0312, Y 13.0208, Z -4.6667, A 0.000, B 0.000, C 0.000 }
gfCNCPoint3[27957] = {X 547.9288, Y 13.8964, Z -4.6667, A 0.000, B 0.000, C 0.000 }
gfCNCPoint3[27958] = {X 547.6442, Y 14.7307, Z -4.6667, A 0.000, B 0.000, C 0.000 }
gfCNCPoint3[27959] = {X 547.1902, Y 15.4863, Z -4.6667, A 0.000, B 0.000, C 0.000 }
gfCNCPoint3[27960] = {X 546.5871, Y 16.1293, Z -4.6667, A 0.000, B 0.000, C 0.000 }
gfCNCPoint3[27961] = {X 546.5038, Y 16.1992, Z -4.6667, A 0.000, B 0.000, C 0.000 }
gfCNCPoint3[27962] = {X 546.5040, Y 40.9897, Z -4.6667, A 0.000, B 0.000, C 0.000 }
gfCNCPoint3[27963] = {X 546.5834, Y 41.0543, Z -4.6667, A 0.000, B 0.000, C 0.000 }
gfCNCPoint3[27964] = {X 547.1893, Y 41.6993, Z -4.6667, A 0.000, B 0.000, C 0.000 }
gfCNCPoint3[27965] = {X 547.6450, Y 42.4578, Z -4.6667, A 0.000, B 0.000, C 0.000 }
gfCNCPoint3[27966] = {X 547.9299, Y 43.2956, Z -4.6667, A 0.000, B 0.000, C 0.000 }
gfCNCPoint3[27967] = {X 548.0313, Y 44.1746, Z -4.6667, A 0.000, B 0.000, C 0.000 }
gfCNCPoint3[27968] = {X 548.0314, Y 45.0002, Z -4.6667, A 0.000, B 0.000, C 0.000 }
gfCNCPoint3[27969] = {X 547.9220, Y 45.9417, Z -4.6667, A 0.000, B 0.000, C 0.000 }
gfCNCPoint3[27970] = {X 547.6024, Y 46.8341, Z -4.6667, A 0.000, B 0.000, C 0.000 }
gfCNCPoint3[27971] = {X 547.0894, Y 47.6311, Z -4.6667, A 0.000, B 0.000, C 0.000 }
gfCNCPoint3[27972] = {X 546.4094, Y 48.2914, Z -4.6667, A 0.000, B 0.000, C 0.000 }
gfCNCPoint3[27973] = {X 545.5977, Y 48.7809, Z -4.6667, A 0.000, B 0.000, C 0.000 }
gfCNCPoint3[27974] = {X 544.6964, Y 49.0741, Z -4.6667, A 0.000, B 0.000, C 0.000 }
gfCNCPoint3[27975] = {X 543.7521, Y 49.1559, Z -4.6667, A 0.000, B 0.000, C 0.000 }
gfCNCPoint3[27976] = {X 523.9616, Y 49.1564, Z -4.6667, A 0.000, B 0.000, C 0.000 }
gfCNCPoint3[27977] = {X 523.4348, Y 49.7889, Z -4.6667, A 0.000, B 0.000, C 0.000 }
gfCNCPoint3[27978] = {X 522.7976, Y 50.3100, Z -4.6667, A 0.000, B 0.000, C 0.000 }
gfCNCPoint3[27979] = {X 522.0730, Y 50.7006, Z -4.6667, A 0.000, B 0.000, C 0.000 }
gfCNCPoint3[27980] = {X 521.2875, Y 50.9467, Z -4.6667, A 0.000, B 0.000, C 0.000 }
gfCNCPoint3[27981] = {X 520.4695, Y 51.0391, Z -4.6667, A 0.000, B 0.000, C 0.000 }
gfCNCPoint3[27982] = {X 519.7998, Y 51.0391, Z -4.6667, A 0.000, B 0.000, C 0.000 }
gfCNCPoint3[27983] = {X 518.8741, Y 50.9348, Z -4.6667, A 0.000, B 0.000, C 0.000 }
gfCNCPoint3[27984] = {X 517.9948, Y 50.6272, Z -4.6667, A 0.000, B 0.000, C 0.000 }
gfCNCPoint3[27985] = {X 517.2061, Y 50.1315, Z -4.6667, A 0.000, B 0.000, C 0.000 }
gfCNCPoint3[27986] = {X 516.5474, Y 49.4728, Z -4.6667, A 0.000, B 0.000, C 0.000 }
gfCNCPoint3[27987] = {X 516.0517, Y 48.6841, Z -4.6667, A 0.000, B 0.000, C 0.000 }
gfCNCPoint3[27988] = {X 515.7441, Y 47.8048, Z -4.6667, A 0.000, B 0.000, C 0.000 }
gfCNCPoint3[27989] = {X 515.6398, Y 46.8791, Z -4.6667, A 0.000, B 0.000, C 0.000 }
gfCNCPoint3[27990] = {X 515.6398, Y 39.9011, Z -4.6667, A 0.000, B 0.000, C 0.000 }
gfCNCPoint3[27991] = {X 515.7429, Y 38.9805, Z -4.6667, A 0.000, B 0.000, C 0.000 }
gfCNCPoint3[27992] = {X 516.0472, Y 38.1056, Z -4.6667, A 0.000, B 0.000, C 0.000 }
gfCNCPoint3[27993] = {X 516.5376, Y 37.3197, Z -4.6667, A 0.000, B 0.000, C 0.000 }
gfCNCPoint3[27994] = {X 517.1897, Y 36.6618, Z -4.6667, A 0.000, B 0.000, C 0.000 }
gfCNCPoint3[27995] = {X 517.9713, Y 36.1645, Z -4.6667, A 0.000, B 0.000, C 0.000 }
gfCNCPoint3[27996] = {X 518.8435, Y 35.8525, Z -4.6667, A 0.000, B 0.000, C 0.000 }
gfCNCPoint3[27997] = {X 519.7631, Y 35.7413, Z -4.6667, A 0.000, B 0.000, C 0.000 }
gfCNCPoint3[27998] = {X 520.5247, Y 35.7415, Z -4.6667, A 0.000, B 0.000, C 0.000 }
gfCNCPoint3[27999] = {X 521.3371, Y 35.8329, Z -4.6667, A 0.000, B 0.000, C 0.000 }
gfCNCPoint3[28000] = {X 522.1159, Y 36.0813, Z -4.6667, A 0.000, B 0.000, C 0.000 }
gfCNCPoint3[28001] = {X 522.8311, Y 36.4773, Z -4.6667, A 0.000, B 0.000, C 0.000 }
gfCNCPoint3[28002] = {X 523.4551, Y 37.0056, Z -4.6667, A 0.000, B 0.000, C 0.000 }
gfCNCPoint3[28003] = {X 523.9637, Y 37.6456, Z -4.6667, A 0.000, B 0.000, C 0.000 }
gfCNCPoint3[28004] = {X 534.7919, Y 37.6461, Z -4.6667, A 0.000, B 0.000, C 0.000 }
gfCNCPoint3[28005] = {X 534.7919, Y 33.8055, Z -4.6667, A 0.000, B 0.000, C 0.000 }
gfCNCPoint3[28006] = {X 530.0216, Y 33.8051, Z -4.6667, A 0.000, B 0.000, C 0.000 }
gfCNCPoint3[28007] = {X 529.9748, Y 33.8793, Z -4.6667, A 0.000, B 0.000, C 0.000 }
gfCNCPoint3[28008] = {X 529.4623, Y 34.4987, Z -4.6667, A 0.000, B 0.000, C 0.000 }
gfCNCPoint3[28009] = {X 528.8402, Y 35.0079, Z -4.6667, A 0.000, B 0.000, C 0.000 }
gfCNCPoint3[28010] = {X 528.1318, Y 35.3880, Z -4.6667, A 0.000, B 0.000, C 0.000 }
gfCNCPoint3[28011] = {X 527.3636, Y 35.6248, Z -4.6667, A 0.000, B 0.000, C 0.000 }
gfCNCPoint3[28012] = {X 526.5641, Y 35.7093, Z -4.6667, A 0.000, B 0.000, C 0.000 }
gfCNCPoint3[28013] = {X 525.8868, Y 35.7095, Z -4.6667, A 0.000, B 0.000, C 0.000 }
gfCNCPoint3[28014] = {X 524.9611, Y 35.6052, Z -4.6667, A 0.000, B 0.000, C 0.000 }
gfCNCPoint3[28015] = {X 524.0818, Y 35.2975, Z -4.6667, A 0.000, B 0.000, C 0.000 }
gfCNCPoint3[28016] = {X 523.2930, Y 34.8019, Z -4.6667, A 0.000, B 0.000, C 0.000 }
gfCNCPoint3[28017] = {X 522.6343, Y 34.1432, Z -4.6667, A 0.000, B 0.000, C 0.000 }
gfCNCPoint3[28018] = {X 522.1387, Y 33.3544, Z -4.6667, A 0.000, B 0.000, C 0.000 }
gfCNCPoint3[28019] = {X 521.8311, Y 32.4751, Z -4.6667, A 0.000, B 0.000, C 0.000 }
gfCNCPoint3[28020] = {X 521.7268, Y 31.5495, Z -4.6667, A 0.000, B 0.000, C 0.000 }
gfCNCPoint3[28021] = {X 521.7268, Y 24.5714, Z -4.6667, A 0.000, B 0.000, C 0.000 }
gfCNCPoint3[28022] = {X 521.8299, Y 23.6507, Z -4.6667, A 0.000, B 0.000, C 0.000 }
gfCNCPoint3[28023] = {X 522.1343, Y 22.7756, Z -4.6667, A 0.000, B 0.000, C 0.000 }
gfCNCPoint3[28024] = {X 522.6248, Y 21.9897, Z -4.6667, A 0.000, B 0.000, C 0.000 }
gfCNCPoint3[28025] = {X 523.2772, Y 21.3317, Z -4.6667, A 0.000, B 0.000, C 0.000 }
gfCNCPoint3[28026] = {X 524.0589, Y 20.8345, Z -4.6667, A 0.000, B 0.000, C 0.000 }
gfCNCPoint3[28027] = {X 524.9313, Y 20.5226, Z -4.6667, A 0.000, B 0.000, C 0.000 }
gfCNCPoint3[28028] = {X 525.8511, Y 20.4116, Z -4.6667, A 0.000, B 0.000, C 0.000 }
gfCNCPoint3[28029] = {X 526.5679, Y 20.4116, Z -4.6667, A 0.000, B 0.000, C 0.000 }
gfCNCPoint3[28030] = {X 527.3789, Y 20.4993, Z -4.6667, A 0.000, B 0.000, C 0.000 }
gfCNCPoint3[28031] = {X 528.1571, Y 20.7435, Z -4.6667, A 0.000, B 0.000, C 0.000 }
gfCNCPoint3[28032] = {X 528.8727, Y 21.1349, Z -4.6667, A 0.000, B 0.000, C 0.000 }
gfCNCPoint3[28033] = {X 529.4982, Y 21.6583, Z -4.6667, A 0.000, B 0.000, C 0.000 }
gfCNCPoint3[28034] = {X 530.0095, Y 22.2938, Z -4.6667, A 0.000, B 0.000, C 0.000 }
gfCNCPoint3[28035] = {X 534.7919, Y 22.2941, Z -4.6667, A 0.000, B 0.000, C 0.000 }
gfCNCPoint3[28036] = {X 534.7919, Y 19.5419, Z -4.6667, A 0.000, B 0.000, C 0.000 }
gfCNCPoint3[28037] = {X 524.1050, Y 19.5416, Z -4.6667, A 0.000, B 0.000, C 0.000 }
gfCNCPoint3[28038] = {X 524.0763, Y 19.5869, Z -4.6667, A 0.000, B 0.000, C 0.000 }
gfCNCPoint3[28039] = {X 523.5639, Y 20.2157, Z -4.6667, A 0.000, B 0.000, C 0.000 }
gfCNCPoint3[28040] = {X 522.9392, Y 20.7331, Z -4.6667, A 0.000, B 0.000, C 0.000 }
gfCNCPoint3[28041] = {X 522.2259, Y 21.1194, Z -4.6667, A 0.000, B 0.000, C 0.000 }
gfCNCPoint3[28042] = {X 521.4513, Y 21.3599, Z -4.6667, A 0.000, B 0.000, C 0.000 }
gfCNCPoint3[28043] = {X 520.6447, Y 21.4456, Z -4.6667, A 0.000, B 0.000, C 0.000 }
gfCNCPoint3[28044] = {X 519.9691, Y 21.4457, Z -4.6667, A 0.000, B 0.000, C 0.000 }
gfCNCPoint3[28045] = {X 519.0434, Y 21.3414, Z -4.6667, A 0.000, B 0.000, C 0.000 }
gfCNCPoint3[28046] = {X 518.1641, Y 21.0337, Z -4.6667, A 0.000, B 0.000, C 0.000 }
gfCNCPoint3[28047] = {X 517.3754, Y 20.5381, Z -4.6667, A 0.000, B 0.000, C 0.000 }
gfCNCPoint3[28048] = {X 516.7167, Y 19.8794, Z -4.6667, A 0.000, B 0.000, C 0.000 }
gfCNCPoint3[28049] = {X 516.2211, Y 19.0907, Z -4.6667, A 0.000, B 0.000, C 0.000 }
gfCNCPoint3[28050] = {X 515.9134, Y 18.2114, Z -4.6667, A 0.000, B 0.000, C 0.000 }
gfCNCPoint3[28051] = {X 515.8091, Y 17.2857, Z -4.6667, A 0.000, B 0.000, C 0.000 }
gfCNCPoint3[28052] = {X 515.8091, Y 10.3077, Z -4.6667, A 0.000, B 0.000, C 0.000 }
gfCNCPoint3[28053] = {X 515.9122, Y 9.3873, Z -4.6667, A 0.000, B 0.000, C 0.000 }
gfCNCPoint3[28054] = {X 516.2164, Y 8.5125, Z -4.6667, A 0.000, B 0.000, C 0.000 }
gfCNCPoint3[28055] = {X 516.7065, Y 7.7267, Z -4.6667, A 0.000, B 0.000, C 0.000 }
gfCNCPoint3[28056] = {X 517.3584, Y 7.0689, Z -4.6667, A 0.000, B 0.000, C 0.000 }
gfCNCPoint3[28057] = {X 518.1397, Y 6.5715, Z -4.6667, A 0.000, B 0.000, C 0.000 }
gfCNCPoint3[28058] = {X 519.0117, Y 6.2594, Z -4.6667, A 0.000, B 0.000, C 0.000 }
gfCNCPoint3[28059] = {X 519.9311, Y 6.1479, Z -4.6667, A 0.000, B 0.000, C 0.000 }
gfCNCPoint3[28060] = {X 520.6487, Y 6.1479, Z -4.6667, A 0.000, B 0.000, C 0.000 }
gfCNCPoint3[28061] = {X 521.4600, Y 6.2353, Z -4.6667, A 0.000, B 0.000, C 0.000 }
gfCNCPoint3[28062] = {X 522.2386, Y 6.4794, Z -4.6667, A 0.000, B 0.000, C 0.000 }
gfCNCPoint3[28063] = {X 522.9546, Y 6.8708, Z -4.6667, A 0.000, B 0.000, C 0.000 }
gfCNCPoint3[28064] = {X 523.5804, Y 7.3944, Z -4.6667, A 0.000, B 0.000, C 0.000 }
gfCNCPoint3[28065] = {X 524.0919, Y 8.0301, Z -4.6667, A 0.000, B 0.000, C 0.000 }
gfCNCPoint3[28066] = {X 533.9636, Y 8.0303, Z -4.6667, A 0.000, B 0.000, C 0.000 }
gfCNCPoint3[28067] = {X 533.9637, Y 4.0303, Z -4.6667, A 0.000, B 0.000, C 0.000 }
gfCNCPoint3[28068] = {X 533.9636, Y 8.1103, Z -4.6667, A 0.000, B 0.000, C 0.000 }
gfCNCPoint3[28069] = {X 543.7532, Y 8.1106, Z -4.6667, A 0.000, B 0.000, C 0.000 }
gfCNCPoint3[28070] = {X 544.6796, Y 8.1907, Z -4.6667, A 0.000, B 0.000, C 0.000 }
gfCNCPoint3[28071] = {X 545.5638, Y 8.4783, Z -4.6667, A 0.000, B 0.000, C 0.000 }
gfCNCPoint3[28072] = {X 546.3601, Y 8.9583, Z -4.6667, A 0.000, B 0.000, C 0.000 }
gfCNCPoint3[28073] = {X 547.0272, Y 9.6060, Z -4.6667, A 0.000, B 0.000, C 0.000 }
gfCNCPoint3[28074] = {X 547.5305, Y 10.3878, Z -4.6667, A 0.000, B 0.000, C 0.000 }
gfCNCPoint3[28075] = {X 547.8440, Y 11.2631, Z -4.6667, A 0.000, B 0.000, C 0.000 }
gfCNCPoint3[28076] = {X 547.9514, Y 12.1867, Z -4.6667, A 0.000, B 0.000, C 0.000 }
gfCNCPoint3[28077] = {X 547.9512, Y 13.0200, Z -4.6667, A 0.000, B 0.000, C 0.000 }
gfCNCPoint3[28078] = {X 547.8508, Y 13.8787, Z -4.6667, A 0.000, B 0.000, C 0.000 }
gfCNCPoint3[28079] = {X 547.5716, Y 14.6970, Z -4.6667, A 0.000, B 0.000, C 0.000 }
gfCNCPoint3[28080] = {X 547.1263, Y 15.4381, Z -4.6667, A 0.000, B 0.000, C 0.000 }
gfCNCPoint3[28081] = {X 546.5349, Y 16.0687, Z -4.6667, A 0.000, B 0.000, C 0.000 }
gfCNCPoint3[28082] = {X 546.4802, Y 16.1150, Z -4.6667, A 0.000, B 0.000, C 0.000 }
gfCNCPoint3[28083] = {X 546.4247, Y 16.1603, Z -4.6667, A 0.000, B 0.000, C 0.000 }
gfCNCPoint3[28084] = {X 546.4240, Y 41.0277, Z -4.6667, A 0.000, B 0.000, C 0.000 }
gfCNCPoint3[28085] = {X 546.5321, Y 41.1157, Z -4.6667, A 0.000, B 0.000, C 0.000 }
gfCNCPoint3[28086] = {X 547.1260, Y 41.7482, Z -4.6667, A 0.000, B 0.000, C 0.000 }
gfCNCPoint3[28087] = {X 547.5726, Y 42.4920, Z -4.6667, A 0.000, B 0.000, C 0.000 }
gfCNCPoint3[28088] = {X 547.8520, Y 43.3134, Z -4.6667, A 0.000, B 0.000, C 0.000 }
gfCNCPoint3[28089] = {X 547.9513, Y 44.1753, Z -4.6667, A 0.000, B 0.000, C 0.000 }
gfCNCPoint3[28090] = {X 547.9514, Y 45.0001, Z -4.6667, A 0.000, B 0.000, C 0.000 }
gfCNCPoint3[28091] = {X 547.8440, Y 45.9237, Z -4.6667, A 0.000, B 0.000, C 0.000 }
gfCNCPoint3[28092] = {X 547.5305, Y 46.7990, Z -4.6667, A 0.000, B 0.000, C 0.000 }
gfCNCPoint3[28093] = {X 547.0272, Y 47.5807, Z -4.6667, A 0.000, B 0.000, C 0.000 }
gfCNCPoint3[28094] = {X 546.3601, Y 48.2284, Z -4.6667, A 0.000, B 0.000, C 0.000 }
gfCNCPoint3[28095] = {X 545.5638, Y 48.7084, Z -4.6667, A 0.000, B 0.000, C 0.000 }
gfCNCPoint3[28096] = {X 544.6796, Y 48.9959, Z -4.6667, A 0.000, B 0.000, C 0.000 }
gfCNCPoint3[28097] = {X 543.7532, Y 49.0759, Z -4.6667, A 0.000, B 0.000, C 0.000 }
gfCNCPoint3[28098] = {X 523.9191, Y 49.0764, Z -4.6667, A 0.000, B 0.000, C 0.000 }
gfCNCPoint3[28099] = {X 523.4024, Y 49.7082, Z -4.6667, A 0.000, B 0.000, C 0.000 }
gfCNCPoint3[28100] = {X 522.7742, Y 50.2292, Z -4.6667, A 0.000, B 0.000, C 0.000 }
gfCNCPoint3[28101] = {X 522.0578, Y 50.6202, Z -4.6667, A 0.000, B 0.000, C 0.000 }
gfCNCPoint3[28102] = {X 521.2797, Y 50.8665, Z -4.6667, A 0.000, B 0.000, C 0.000 }
gfCNCPoint3[28103] = {X 520.4688, Y 50.9591, Z -4.6667, A 0.000, B 0.000, C 0.000 }
gfCNCPoint3[28104] = {X 519.7998, Y 50.9591, Z -4.6667, A 0.000, B 0.000, C 0.000 }
gfCNCPoint3[28105] = {X 518.8919, Y 50.8568, Z -4.6667, A 0.000, B 0.000, C 0.000 }
gfCNCPoint3[28106] = {X 518.0295, Y 50.5551, Z -4.6667, A 0.000, B 0.000, C 0.000 }
gfCNCPoint3[28107] = {X 517.2559, Y 50.0690, Z -4.6667, A 0.000, B 0.000, C 0.000 }
gfCNCPoint3[28108] = {X 516.6099, Y 49.4230, Z -4.6667, A 0.000, B 0.000, C 0.000 }
gfCNCPoint3[28109] = {X 516.1238, Y 48.6494, Z -4.6667, A 0.000, B 0.000, C 0.000 }
gfCNCPoint3[28110] = {X 515.8221, Y 47.7870, Z -4.6667, A 0.000, B 0.000, C 0.000 }
gfCNCPoint3[28111] = {X 515.7198, Y 46.8791, Z -4.6667, A 0.000, B 0.000, C 0.000 }
gfCNCPoint3[28112] = {X 515.7198, Y 39.9011, Z -4.6667, A 0.000, B 0.000, C 0.000 }
gfCNCPoint3[28113] = {X 515.8209, Y 38.9982, Z -4.6667, A 0.000, B 0.000, C 0.000 }
gfCNCPoint3[28114] = {X 516.1194, Y 38.1401, Z -4.6667, A 0.000, B 0.000, C 0.000 }
gfCNCPoint3[28115] = {X 516.6003, Y 37.3693, Z -4.6667, A 0.000, B 0.000, C 0.000 }
gfCNCPoint3[28116] = {X 517.2399, Y 36.7241, Z -4.6667, A 0.000, B 0.000, C 0.000 }
gfCNCPoint3[28117] = {X 518.0064, Y 36.2364, Z -4.6667, A 0.000, B 0.000, C 0.000 }
gfCNCPoint3[28118] = {X 518.8619, Y 35.9304, Z -4.6667, A 0.000, B 0.000, C 0.000 }
gfCNCPoint3[28119] = {X 519.7638, Y 35.8213, Z -4.6667, A 0.000, B 0.000, C 0.000 }
gfCNCPoint3[28120] = {X 520.5236, Y 35.8215, Z -4.6667, A 0.000, B 0.000, C 0.000 }
gfCNCPoint3[28121] = {X 521.3289, Y 35.9129, Z -4.6667, A 0.000, B 0.000, C 0.000 }
gfCNCPoint3[28122] = {X 522.1002, Y 36.1617, Z -4.6667, A 0.000, B 0.000, C 0.000 }
gfCNCPoint3[28123] = {X 522.8071, Y 36.5581, Z -4.6667, A 0.000, B 0.000, C 0.000 }
gfCNCPoint3[28124] = {X 523.4217, Y 37.0863, Z -4.6667, A 0.000, B 0.000, C 0.000 }
gfCNCPoint3[28125] = {X 523.9198, Y 37.7256, Z -4.6667, A 0.000, B 0.000, C 0.000 }
gfCNCPoint3[28126] = {X 534.8719, Y 37.7261, Z -4.6667, A 0.000, B 0.000, C 0.000 }
gfCNCPoint3[28127] = {X 534.8719, Y 33.7255, Z -4.6667, A 0.000, B 0.000, C 0.000 }
gfCNCPoint3[28128] = {X 529.9775, Y 33.7251, Z -4.6667, A 0.000, B 0.000, C 0.000 }
gfCNCPoint3[28129] = {X 529.9071, Y 33.8366, Z -4.6667, A 0.000, B 0.000, C 0.000 }
gfCNCPoint3[28130] = {X 529.2612, Y 34.5790, Z -4.6667, A 0.000, B 0.000, C 0.000 }
gfCNCPoint3[28131] = {X 528.4563, Y 35.1452, Z -4.6667, A 0.000, B 0.000, C 0.000 }
gfCNCPoint3[28132] = {X 527.5392, Y 35.5023, Z -4.6667, A 0.000, B 0.000, C 0.000 }
gfCNCPoint3[28133] = {X 526.5634, Y 35.6293, Z -4.6667, A 0.000, B 0.000, C 0.000 }
gfCNCPoint3[28134] = {X 525.8868, Y 35.6295, Z -4.6667, A 0.000, B 0.000, C 0.000 }
gfCNCPoint3[28135] = {X 524.9789, Y 35.5272, Z -4.6667, A 0.000, B 0.000, C 0.000 }
gfCNCPoint3[28136] = {X 524.1165, Y 35.2254, Z -4.6667, A 0.000, B 0.000, C 0.000 }
gfCNCPoint3[28137] = {X 523.3429, Y 34.7393, Z -4.6667, A 0.000, B 0.000, C 0.000 }
gfCNCPoint3[28138] = {X 522.6969, Y 34.0933, Z -4.6667, A 0.000, B 0.000, C 0.000 }
gfCNCPoint3[28139] = {X 522.2108, Y 33.3197, Z -4.6667, A 0.000, B 0.000, C 0.000 }
gfCNCPoint3[28140] = {X 521.9091, Y 32.4573, Z -4.6667, A 0.000, B 0.000, C 0.000 }
gfCNCPoint3[28141] = {X 521.8068, Y 31.5495, Z -4.6667, A 0.000, B 0.000, C 0.000 }
gfCNCPoint3[28142] = {X 521.8068, Y 24.5714, Z -4.6667, A 0.000, B 0.000, C 0.000 }
gfCNCPoint3[28143] = {X 521.9079, Y 23.6684, Z -4.6667, A 0.000, B 0.000, C 0.000 }
gfCNCPoint3[28144] = {X 522.2065, Y 22.8102, Z -4.6667, A 0.000, B 0.000, C 0.000 }
gfCNCPoint3[28145] = {X 522.6876, Y 22.0393, Z -4.6667, A 0.000, B 0.000, C 0.000 }
gfCNCPoint3[28146] = {X 523.3273, Y 21.3940, Z -4.6667, A 0.000, B 0.000, C 0.000 }
gfCNCPoint3[28147] = {X 524.0941, Y 20.9064, Z -4.6667, A 0.000, B 0.000, C 0.000 }
gfCNCPoint3[28148] = {X 524.9497, Y 20.6005, Z -4.6667, A 0.000, B 0.000, C 0.000 }
gfCNCPoint3[28149] = {X 525.8518, Y 20.4916, Z -4.6667, A 0.000, B 0.000, C 0.000 }
gfCNCPoint3[28150] = {X 526.5672, Y 20.4916, Z -4.6667, A 0.000, B 0.000, C 0.000 }
gfCNCPoint3[28151] = {X 527.3709, Y 20.5794, Z -4.6667, A 0.000, B 0.000, C 0.000 }
gfCNCPoint3[28152] = {X 528.1416, Y 20.8239, Z -4.6667, A 0.000, B 0.000, C 0.000 }
gfCNCPoint3[28153] = {X 528.8489, Y 21.2156, Z -4.6667, A 0.000, B 0.000, C 0.000 }
gfCNCPoint3[28154] = {X 529.4651, Y 21.7391, Z -4.6667, A 0.000, B 0.000, C 0.000 }
gfCNCPoint3[28155] = {X 529.9660, Y 22.3738, Z -4.6667, A 0.000, B 0.000, C 0.000 }
gfCNCPoint3[28156] = {X 534.8719, Y 22.3741, Z -4.6667, A 0.000, B 0.000, C 0.000 }
gfCNCPoint3[28157] = {X 534.8719, Y 19.4619, Z -4.6667, A 0.000, B 0.000, C 0.000 }
gfCNCPoint3[28158] = {X 524.0609, Y 19.4616, Z -4.6667, A 0.000, B 0.000, C 0.000 }
gfCNCPoint3[28159] = {X 524.0087, Y 19.5442, Z -4.6667, A 0.000, B 0.000, C 0.000 }
gfCNCPoint3[28160] = {X 523.5061, Y 20.1604, Z -4.6667, A 0.000, B 0.000, C 0.000 }
gfCNCPoint3[28161] = {X 522.8935, Y 20.6674, Z -4.6667, A 0.000, B 0.000, C 0.000 }
gfCNCPoint3[28162] = {X 522.1942, Y 21.0459, Z -4.6667, A 0.000, B 0.000, C 0.000 }
gfCNCPoint3[28163] = {X 521.4348, Y 21.2816, Z -4.6667, A 0.000, B 0.000, C 0.000 }
gfCNCPoint3[28164] = {X 520.6440, Y 21.3656, Z -4.6667, A 0.000, B 0.000, C 0.000 }
gfCNCPoint3[28165] = {X 519.9691, Y 21.3657, Z -4.6667, A 0.000, B 0.000, C 0.000 }
gfCNCPoint3[28166] = {X 519.0612, Y 21.2634, Z -4.6667, A 0.000, B 0.000, C 0.000 }
gfCNCPoint3[28167] = {X 518.1989, Y 20.9617, Z -4.6667, A 0.000, B 0.000, C 0.000 }
gfCNCPoint3[28168] = {X 517.4253, Y 20.4756, Z -4.6667, A 0.000, B 0.000, C 0.000 }
gfCNCPoint3[28169] = {X 516.7792, Y 19.8296, Z -4.6667, A 0.000, B 0.000, C 0.000 }
gfCNCPoint3[28170] = {X 516.2932, Y 19.0560, Z -4.6667, A 0.000, B 0.000, C 0.000 }
gfCNCPoint3[28171] = {X 515.9914, Y 18.1936, Z -4.6667, A 0.000, B 0.000, C 0.000 }
gfCNCPoint3[28172] = {X 515.8891, Y 17.2857, Z -4.6667, A 0.000, B 0.000, C 0.000 }
gfCNCPoint3[28173] = {X 515.8891, Y 10.3077, Z -4.6667, A 0.000, B 0.000, C 0.000 }
gfCNCPoint3[28174] = {X 515.9902, Y 9.4050, Z -4.6667, A 0.000, B 0.000, C 0.000 }
gfCNCPoint3[28175] = {X 516.2885, Y 8.5471, Z -4.6667, A 0.000, B 0.000, C 0.000 }
gfCNCPoint3[28176] = {X 516.7693, Y 7.7764, Z -4.6667, A 0.000, B 0.000, C 0.000 }
gfCNCPoint3[28177] = {X 517.4086, Y 7.1312, Z -4.6667, A 0.000, B 0.000, C 0.000 }
gfCNCPoint3[28178] = {X 518.1749, Y 6.6434, Z -4.6667, A 0.000, B 0.000, C 0.000 }
gfCNCPoint3[28179] = {X 519.0301, Y 6.3372, Z -4.6667, A 0.000, B 0.000, C 0.000 }
gfCNCPoint3[28180] = {X 519.9318, Y 6.2279, Z -4.6667, A 0.000, B 0.000, C 0.000 }
gfCNCPoint3[28181] = {X 520.6480, Y 6.2279, Z -4.6667, A 0.000, B 0.000, C 0.000 }
gfCNCPoint3[28182] = {X 521.4521, Y 6.3154, Z -4.6667, A 0.000, B 0.000, C 0.000 }
gfCNCPoint3[28183] = {X 522.2231, Y 6.5598, Z -4.6667, A 0.000, B 0.000, C 0.000 }
gfCNCPoint3[28184] = {X 522.9308, Y 6.9515, Z -4.6667, A 0.000, B 0.000, C 0.000 }
gfCNCPoint3[28185] = {X 523.5473, Y 7.4752, Z -4.6667, A 0.000, B 0.000, C 0.000 }
gfCNCPoint3[28186] = {X 524.0484, Y 8.1101, Z -4.6667, A 0.000, B 0.000, C 0.000 }
gfCNCPoint3[28187] = {X 533.9636, Y 8.1103, Z -4.6667, A 0.000, B 0.000, C 0.000 }
gfCNCPoint3[28188] = {X 533.9637, Y 4.1103, Z -4.6667, A 0.000, B 0.000, C 0.000 }
gfCNCPoint3[28189] = {X 533.9636, Y 8.1903, Z -4.6667, A 0.000, B 0.000, C 0.000 }
gfCNCPoint3[28190] = {X 543.7544, Y 8.1906, Z -4.6667, A 0.000, B 0.000, C 0.000 }
gfCNCPoint3[28191] = {X 544.6627, Y 8.2689, Z -4.6667, A 0.000, B 0.000, C 0.000 }
gfCNCPoint3[28192] = {X 545.5298, Y 8.5507, Z -4.6667, A 0.000, B 0.000, C 0.000 }
gfCNCPoint3[28193] = {X 546.3107, Y 9.0213, Z -4.6667, A 0.000, B 0.000, C 0.000 }
gfCNCPoint3[28194] = {X 546.9650, Y 9.6563, Z -4.6667, A 0.000, B 0.000, C 0.000 }
gfCNCPoint3[28195] = {X 547.4586, Y 10.4229, Z -4.6667, A 0.000, B 0.000, C 0.000 }
gfCNCPoint3[28196] = {X 547.7661, Y 11.2812, Z -4.6667, A 0.000, B 0.000, C 0.000 }
gfCNCPoint3[28197] = {X 547.8714, Y 12.1869, Z -4.6667, A 0.000, B 0.000, C 0.000 }
gfCNCPoint3[28198] = {X 547.8712, Y 13.0192, Z -4.6667, A 0.000, B 0.000, C 0.000 }
gfCNCPoint3[28199] = {X 547.7727, Y 13.8611, Z -4.6667, A 0.000, B 0.000, C 0.000 }
gfCNCPoint3[28200] = {X 547.4991, Y 14.6633, Z -4.6667, A 0.000, B 0.000, C 0.000 }
gfCNCPoint3[28201] = {X 547.0625, Y 15.3898, Z -4.6667, A 0.000, B 0.000, C 0.000 }
gfCNCPoint3[28202] = {X 546.4827, Y 16.0081, Z -4.6667, A 0.000, B 0.000, C 0.000 }
gfCNCPoint3[28203] = {X 546.4149, Y 16.0652, Z -4.6667, A 0.000, B 0.000, C 0.000 }
gfCNCPoint3[28204] = {X 546.3458, Y 16.1209, Z -4.6667, A 0.000, B 0.000, C 0.000 }
gfCNCPoint3[28205] = {X 546.3438, Y 16.3111, Z -4.6667, A 0.000, B 0.000, C 0.000 }
gfCNCPoint3[28206] = {X 546.3440, Y 41.0658, Z -4.6667, A 0.000, B 0.000, C 0.000 }
gfCNCPoint3[28207] = {X 546.4829, Y 41.1789, Z -4.6667, A 0.000, B 0.000, C 0.000 }
gfCNCPoint3[28208] = {X 547.0689, Y 41.8054, Z -4.6667, A 0.000, B 0.000, C 0.000 }
gfCNCPoint3[28209] = {X 547.5078, Y 42.5424, Z -4.6667, A 0.000, B 0.000, C 0.000 }
gfCNCPoint3[28210] = {X 547.7795, Y 43.3560, Z -4.6667, A 0.000, B 0.000, C 0.000 }
gfCNCPoint3[28211] = {X 547.8714, Y 44.2089, Z -4.6667, A 0.000, B 0.000, C 0.000 }
gfCNCPoint3[28212] = {X 547.8714, Y 45.0000, Z -4.6667, A 0.000, B 0.000, C 0.000 }
gfCNCPoint3[28213] = {X 547.7661, Y 45.9056, Z -4.6667, A 0.000, B 0.000, C 0.000 }
gfCNCPoint3[28214] = {X 547.4586, Y 46.7639, Z -4.6667, A 0.000, B 0.000, C 0.000 }
gfCNCPoint3[28215] = {X 546.9650, Y 47.5304, Z -4.6667, A 0.000, B 0.000, C 0.000 }
gfCNCPoint3[28216] = {X 546.3107, Y 48.1654, Z -4.6667, A 0.000, B 0.000, C 0.000 }
gfCNCPoint3[28217] = {X 545.5298, Y 48.6360, Z -4.6667, A 0.000, B 0.000, C 0.000 }
gfCNCPoint3[28218] = {X 544.6627, Y 48.9177, Z -4.6667, A 0.000, B 0.000, C 0.000 }
gfCNCPoint3[28219] = {X 543.7544, Y 48.9959, Z -4.6667, A 0.000, B 0.000, C 0.000 }
gfCNCPoint3[28220] = {X 523.8761, Y 48.9964, Z -4.6667, A 0.000, B 0.000, C 0.000 }
gfCNCPoint3[28221] = {X 523.3697, Y 49.6274, Z -4.6667, A 0.000, B 0.000, C 0.000 }
gfCNCPoint3[28222] = {X 522.7507, Y 50.1484, Z -4.6667, A 0.000, B 0.000, C 0.000 }
gfCNCPoint3[28223] = {X 522.0425, Y 50.5397, Z -4.6667, A 0.000, B 0.000, C 0.000 }
gfCNCPoint3[28224] = {X 521.2719, Y 50.7864, Z -4.6667, A 0.000, B 0.000, C 0.000 }
gfCNCPoint3[28225] = {X 520.4681, Y 50.8791, Z -4.6667, A 0.000, B 0.000, C 0.000 }
gfCNCPoint3[28226] = {X 519.7998, Y 50.8791, Z -4.6667, A 0.000, B 0.000, C 0.000 }
gfCNCPoint3[28227] = {X 518.9097, Y 50.7788, Z -4.6667, A 0.000, B 0.000, C 0.000 }
gfCNCPoint3[28228] = {X 518.0642, Y 50.4830, Z -4.6667, A 0.000, B 0.000, C 0.000 }
gfCNCPoint3[28229] = {X 517.3058, Y 50.0064, Z -4.6667, A 0.000, B 0.000, C 0.000 }
gfCNCPoint3[28230] = {X 516.6724, Y 49.3731, Z -4.6667, A 0.000, B 0.000, C 0.000 }
gfCNCPoint3[28231] = {X 516.1959, Y 48.6147, Z -4.6667, A 0.000, B 0.000, C 0.000 }
gfCNCPoint3[28232] = {X 515.9001, Y 47.7692, Z -4.6667, A 0.000, B 0.000, C 0.000 }
gfCNCPoint3[28233] = {X 515.7998, Y 46.8791, Z -4.6667, A 0.000, B 0.000, C 0.000 }
gfCNCPoint3[28234] = {X 515.7998, Y 39.9011, Z -4.6667, A 0.000, B 0.000, C 0.000 }
gfCNCPoint3[28235] = {X 515.9001, Y 39.0110, Z -4.6667, A 0.000, B 0.000, C 0.000 }
gfCNCPoint3[28236] = {X 516.1959, Y 38.1655, Z -4.6667, A 0.000, B 0.000, C 0.000 }
gfCNCPoint3[28237] = {X 516.6725, Y 37.4071, Z -4.6667, A 0.000, B 0.000, C 0.000 }
gfCNCPoint3[28238] = {X 517.3058, Y 36.7737, Z -4.6667, A 0.000, B 0.000, C 0.000 }
gfCNCPoint3[28239] = {X 518.0643, Y 36.2972, Z -4.6667, A 0.000, B 0.000, C 0.000 }
gfCNCPoint3[28240] = {X 518.9097, Y 36.0014, Z -4.6667, A 0.000, B 0.000, C 0.000 }
gfCNCPoint3[28241] = {X 519.7998, Y 35.9011, Z -4.6667, A 0.000, B 0.000, C 0.000 }
gfCNCPoint3[28242] = {X 520.5225, Y 35.9015, Z -4.6667, A 0.000, B 0.000, C 0.000 }
gfCNCPoint3[28243] = {X 521.3206, Y 35.9930, Z -4.6667, A 0.000, B 0.000, C 0.000 }
gfCNCPoint3[28244] = {X 522.0843, Y 36.2421, Z -4.6667, A 0.000, B 0.000, C 0.000 }
gfCNCPoint3[28245] = {X 522.7828, Y 36.6388, Z -4.6667, A 0.000, B 0.000, C 0.000 }
gfCNCPoint3[28246] = {X 523.3880, Y 37.1671, Z -4.6667, A 0.000, B 0.000, C 0.000 }
gfCNCPoint3[28247] = {X 523.8754, Y 37.8056, Z -4.6667, A 0.000, B 0.000, C 0.000 }
gfCNCPoint3[28248] = {X 534.9519, Y 37.8061, Z -4.6667, A 0.000, B 0.000, C 0.000 }
gfCNCPoint3[28249] = {X 534.9519, Y 34.0455, Z -4.6667, A 0.000, B 0.000, C 0.000 }
gfCNCPoint3[28250] = {X 534.9524, Y 33.6455, Z -4.6667, A 0.000, B 0.000, C 0.000 }
gfCNCPoint3[28251] = {X 529.9334, Y 33.6451, Z -4.6667, A 0.000, B 0.000, C 0.000 }
gfCNCPoint3[28252] = {X 529.8228, Y 33.8182, Z -4.6667, A 0.000, B 0.000, C 0.000 }
gfCNCPoint3[28253] = {X 529.1833, Y 34.5414, Z -4.6667, A 0.000, B 0.000, C 0.000 }
gfCNCPoint3[28254] = {X 528.3891, Y 35.0903, Z -4.6667, A 0.000, B 0.000, C 0.000 }
gfCNCPoint3[28255] = {X 527.4866, Y 35.4330, Z -4.6667, A 0.000, B 0.000, C 0.000 }
gfCNCPoint3[28256] = {X 526.5283, Y 35.5495, Z -4.6667, A 0.000, B 0.000, C 0.000 }
gfCNCPoint3[28257] = {X 525.8868, Y 35.5495, Z -4.6667, A 0.000, B 0.000, C 0.000 }
gfCNCPoint3[28258] = {X 524.9967, Y 35.4492, Z -4.6667, A 0.000, B 0.000, C 0.000 }
gfCNCPoint3[28259] = {X 524.1512, Y 35.1533, Z -4.6667, A 0.000, B 0.000, C 0.000 }
gfCNCPoint3[28260] = {X 523.3928, Y 34.6768, Z -4.6667, A 0.000, B 0.000, C 0.000 }
gfCNCPoint3[28261] = {X 522.7594, Y 34.0434, Z -4.6667, A 0.000, B 0.000, C 0.000 }
gfCNCPoint3[28262] = {X 522.2829, Y 33.2850, Z -4.6667, A 0.000, B 0.000, C 0.000 }
gfCNCPoint3[28263] = {X 521.9870, Y 32.4395, Z -4.6667, A 0.000, B 0.000, C 0.000 }
gfCNCPoint3[28264] = {X 521.8868, Y 31.5495, Z -4.6667, A 0.000, B 0.000, C 0.000 }
gfCNCPoint3[28265] = {X 521.8868, Y 24.5714, Z -4.6667, A 0.000, B 0.000, C 0.000 }
gfCNCPoint3[28266] = {X 521.9870, Y 23.6813, Z -4.6667, A 0.000, B 0.000, C 0.000 }
gfCNCPoint3[28267] = {X 522.2829, Y 22.8359, Z -4.6667, A 0.000, B 0.000, C 0.000 }
gfCNCPoint3[28268] = {X 522.7594, Y 22.0775, Z -4.6667, A 0.000, B 0.000, C 0.000 }
gfCNCPoint3[28269] = {X 523.3928, Y 21.4441, Z -4.6667, A 0.000, B 0.000, C 0.000 }
gfCNCPoint3[28270] = {X 524.1512, Y 20.9675, Z -4.6667, A 0.000, B 0.000, C 0.000 }
gfCNCPoint3[28271] = {X 524.9967, Y 20.6717, Z -4.6667, A 0.000, B 0.000, C 0.000 }
gfCNCPoint3[28272] = {X 525.8868, Y 20.5714, Z -4.6667, A 0.000, B 0.000, C 0.000 }
gfCNCPoint3[28273] = {X 526.5664, Y 20.5716, Z -4.6667, A 0.000, B 0.000, C 0.000 }
gfCNCPoint3[28274] = {X 527.3630, Y 20.6595, Z -4.6667, A 0.000, B 0.000, C 0.000 }
gfCNCPoint3[28275] = {X 528.1260, Y 20.9043, Z -4.6667, A 0.000, B 0.000, C 0.000 }
gfCNCPoint3[28276] = {X 528.8249, Y 21.2964, Z -4.6667, A 0.000, B 0.000, C 0.000 }
gfCNCPoint3[28277] = {X 529.4317, Y 21.8199, Z -4.6667, A 0.000, B 0.000, C 0.000 }
gfCNCPoint3[28278] = {X 529.9219, Y 22.4538, Z -4.6667, A 0.000, B 0.000, C 0.000 }
gfCNCPoint3[28279] = {X 534.9519, Y 22.4541, Z -4.6667, A 0.000, B 0.000, C 0.000 }
gfCNCPoint3[28280] = {X 534.9519, Y 19.7819, Z -4.6667, A 0.000, B 0.000, C 0.000 }
gfCNCPoint3[28281] = {X 534.9525, Y 19.3819, Z -4.6667, A 0.000, B 0.000, C 0.000 }
gfCNCPoint3[28282] = {X 524.0168, Y 19.3816, Z -4.6667, A 0.000, B 0.000, C 0.000 }
gfCNCPoint3[28283] = {X 523.9050, Y 19.5547, Z -4.6667, A 0.000, B 0.000, C 0.000 }
gfCNCPoint3[28284] = {X 523.2655, Y 20.2778, Z -4.6667, A 0.000, B 0.000, C 0.000 }
gfCNCPoint3[28285] = {X 522.4714, Y 20.8266, Z -4.6667, A 0.000, B 0.000, C 0.000 }
gfCNCPoint3[28286] = {X 521.5690, Y 21.1693, Z -4.6667, A 0.000, B 0.000, C 0.000 }
gfCNCPoint3[28287] = {X 520.6107, Y 21.2857, Z -4.6667, A 0.000, B 0.000, C 0.000 }
gfCNCPoint3[28288] = {X 519.9691, Y 21.2857, Z -4.6667, A 0.000, B 0.000, C 0.000 }
gfCNCPoint3[28289] = {X 519.0790, Y 21.1854, Z -4.6667, A 0.000, B 0.000, C 0.000 }
gfCNCPoint3[28290] = {X 518.2336, Y 20.8896, Z -4.6667, A 0.000, B 0.000, C 0.000 }
gfCNCPoint3[28291] = {X 517.4751, Y 20.4130, Z -4.6667, A 0.000, B 0.000, C 0.000 }
gfCNCPoint3[28292] = {X 516.8418, Y 19.7797, Z -4.6667, A 0.000, B 0.000, C 0.000 }
gfCNCPoint3[28293] = {X 516.3652, Y 19.0212, Z -4.6667, A 0.000, B 0.000, C 0.000 }
gfCNCPoint3[28294] = {X 516.0694, Y 18.1758, Z -4.6667, A 0.000, B 0.000, C 0.000 }
gfCNCPoint3[28295] = {X 515.9691, Y 17.2857, Z -4.6667, A 0.000, B 0.000, C 0.000 }
gfCNCPoint3[28296] = {X 515.9691, Y 10.3077, Z -4.6667, A 0.000, B 0.000, C 0.000 }
gfCNCPoint3[28297] = {X 516.0694, Y 9.4176, Z -4.6667, A 0.000, B 0.000, C 0.000 }
gfCNCPoint3[28298] = {X 516.3652, Y 8.5721, Z -4.6667, A 0.000, B 0.000, C 0.000 }
gfCNCPoint3[28299] = {X 516.8418, Y 7.8137, Z -4.6667, A 0.000, B 0.000, C 0.000 }
gfCNCPoint3[28300] = {X 517.4752, Y 7.1803, Z -4.6667, A 0.000, B 0.000, C 0.000 }
gfCNCPoint3[28301] = {X 518.2336, Y 6.7038, Z -4.6667, A 0.000, B 0.000, C 0.000 }
gfCNCPoint3[28302] = {X 519.0791, Y 6.4080, Z -4.6667, A 0.000, B 0.000, C 0.000 }
gfCNCPoint3[28303] = {X 519.9692, Y 6.3077, Z -4.6667, A 0.000, B 0.000, C 0.000 }
gfCNCPoint3[28304] = {X 520.6473, Y 6.3079, Z -4.6667, A 0.000, B 0.000, C 0.000 }
gfCNCPoint3[28305] = {X 521.4441, Y 6.3955, Z -4.6667, A 0.000, B 0.000, C 0.000 }
gfCNCPoint3[28306] = {X 522.2075, Y 6.6402, Z -4.6667, A 0.000, B 0.000, C 0.000 }
gfCNCPoint3[28307] = {X 522.9068, Y 7.0323, Z -4.6667, A 0.000, B 0.000, C 0.000 }
gfCNCPoint3[28308] = {X 523.5139, Y 7.5559, Z -4.6667, A 0.000, B 0.000, C 0.000 }
gfCNCPoint3[28309] = {X 524.0043, Y 8.1901, Z -4.6667, A 0.000, B 0.000, C 0.000 }
gfCNCPoint3[28310] = {X 533.9636, Y 8.1903, Z -4.6667, A 0.000, B 0.000, C 0.000 }
gfCNCPoint3[28311] = {X 533.9637, Y 4.1103, Z -4.6667, A 0.000, B 0.000, C 0.000 }
gfCNCPoint3[28312] = {X 533.9637, Y 4.1103, Z -1.6667, A 0.000, B 0.000, C 0.000 }
gfCNCPoint3[28313] = {X 533.9637, Y 4.1103, Z 11.0000, A 0.000, B 0.000, C 0.000 }
gfCNCPoint3[28314] = {X 419.6141, Y 26.5283, Z 11.0000, A 0.000, B 0.000, C 0.000 }
gfCNCPoint3[28315] = {X 419.6141, Y 26.5283, Z -1.6667, A 0.000, B 0.000, C 0.000 }
gfCNCPoint3[28316] = {X 419.6141, Y 26.5283, Z -4.6667, A 0.000, B 0.000, C 0.000 }
gfCNCPoint3[28317] = {X 416.1507, Y 24.3717, Z -4.6667, A 0.000, B 0.000, C 0.000 }
gfCNCPoint3[28318] = {X 411.5469, Y 31.7651, Z -4.6667, A 0.000, B 0.000, C 0.000 }
gfCNCPoint3[28319] = {X 411.5476, Y 40.8980, Z -4.6667, A 0.000, B 0.000, C 0.000 }
gfCNCPoint3[28320] = {X 412.1858, Y 41.5838, Z -4.6667, A 0.000, B 0.000, C 0.000 }
gfCNCPoint3[28321] = {X 412.6659, Y 42.3883, Z -4.6667, A 0.000, B 0.000, C 0.000 }
gfCNCPoint3[28322] = {X 412.9667, Y 43.2755, Z -4.6667, A 0.000, B 0.000, C 0.000 }
gfCNCPoint3[28323] = {X 413.0747, Y 44.2061, Z -4.6667, A 0.000, B 0.000, C 0.000 }
gfCNCPoint3[28324] = {X 413.0747, Y 45.0002, Z -4.6667, A 0.000, B 0.000, C 0.000 }
gfCNCPoint3[28325] = {X 412.9663, Y 45.9614, Z -4.6667, A 0.000, B 0.000, C 0.000 }
gfCNCPoint3[28326] = {X 412.6468, Y 46.8745, Z -4.6667, A 0.000, B 0.000, C 0.000 }
gfCNCPoint3[28327] = {X 412.1321, Y 47.6935, Z -4.6667, A 0.000, B 0.000, C 0.000 }
gfCNCPoint3[28328] = {X 411.4481, Y 48.3776, Z -4.6667, A 0.000, B 0.000, C 0.000 }
gfCNCPoint3[28329] = {X 410.6290, Y 48.8922, Z -4.6667, A 0.000, B 0.000, C 0.000 }
gfCNCPoint3[28330] = {X 409.7159, Y 49.2117, Z -4.6667, A 0.000, B 0.000, C 0.000 }
gfCNCPoint3[28331] = {X 408.7547, Y 49.3200, Z -4.6667, A 0.000, B 0.000, C 0.000 }
gfCNCPoint3[28332] = {X 402.3112, Y 49.3200, Z -4.6667, A 0.000, B 0.000, C 0.000 }
gfCNCPoint3[28333] = {X 401.3546, Y 49.2127, Z -4.6667, A 0.000, B 0.000, C 0.000 }
gfCNCPoint3[28334] = {X 400.4455, Y 48.8963, Z -4.6667, A 0.000, B 0.000, C 0.000 }
gfCNCPoint3[28335] = {X 399.6290, Y 48.3864, Z -4.6667, A 0.000, B 0.000, C 0.000 }
gfCNCPoint3[28336] = {X 398.9457, Y 47.7084, Z -4.6667, A 0.000, B 0.000, C 0.000 }
gfCNCPoint3[28337] = {X 398.4295, Y 46.8959, Z -4.6667, A 0.000, B 0.000, C 0.000 }
gfCNCPoint3[28338] = {X 398.1060, Y 45.9892, Z -4.6667, A 0.000, B 0.000, C 0.000 }
gfCNCPoint3[28339] = {X 397.9913, Y 45.0335, Z -4.6667, A 0.000, B 0.000, C 0.000 }
gfCNCPoint3[28340] = {X 397.9916, Y 44.1528, Z -4.6667, A 0.000, B 0.000, C 0.000 }
gfCNCPoint3[28341] = {X 398.1015, Y 43.2391, Z -4.6667, A 0.000, B 0.000, C 0.000 }
gfCNCPoint3[28342] = {X 398.4024, Y 42.3694, Z -4.6667, A 0.000, B 0.000, C 0.000 }
gfCNCPoint3[28343] = {X 398.8807, Y 41.5832, Z -4.6667, A 0.000, B 0.000, C 0.000 }
gfCNCPoint3[28344] = {X 399.5147, Y 40.9161, Z -4.6667, A 0.000, B 0.000, C 0.000 }
gfCNCPoint3[28345] = {X 399.4729, Y 31.6004, Z -4.6667, A 0.000, B 0.000, C 0.000 }
gfCNCPoint3[28346] = {X 393.5154, Y 21.2406, Z -4.6667, A 0.000, B 0.000, C 0.000 }
gfCNCPoint3[28347] = {X 392.6279, Y 19.7309, Z -4.6667, A 0.000, B 0.000, C 0.000 }
gfCNCPoint3[28348] = {X 391.7118, Y 18.2384, Z -4.6667, A 0.000, B 0.000, C 0.000 }
gfCNCPoint3[28349] = {X 391.2299, Y 17.5686, Z -4.6667, A 0.000, B 0.000, C 0.000 }
gfCNCPoint3[28350] = {X 390.6670, Y 16.9652, Z -4.6667, A 0.000, B 0.000, C 0.000 }
gfCNCPoint3[28351] = {X 389.7902, Y 16.4729, Z -4.6667, A 0.000, B 0.000, C 0.000 }
gfCNCPoint3[28352] = {X 389.0511, Y 15.7911, Z -4.6667, A 0.000, B 0.000, C 0.000 }
gfCNCPoint3[28353] = {X 388.4896, Y 14.9570, Z -4.6667, A 0.000, B 0.000, C 0.000 }
gfCNCPoint3[28354] = {X 388.1361, Y 14.0156, Z -4.6667, A 0.000, B 0.000, C 0.000 }
gfCNCPoint3[28355] = {X 388.0098, Y 13.0180, Z -4.6667, A 0.000, B 0.000, C 0.000 }
gfCNCPoint3[28356] = {X 388.0096, Y 12.1868, Z -4.6667, A 0.000, B 0.000, C 0.000 }
gfCNCPoint3[28357] = {X 388.1179, Y 11.2255, Z -4.6667, A 0.000, B 0.000, C 0.000 }
gfCNCPoint3[28358] = {X 388.4374, Y 10.3125, Z -4.6667, A 0.000, B 0.000, C 0.000 }
gfCNCPoint3[28359] = {X 388.9521, Y 9.4933, Z -4.6667, A 0.000, B 0.000, C 0.000 }
gfCNCPoint3[28360] = {X 389.6361, Y 8.8093, Z -4.6667, A 0.000, B 0.000, C 0.000 }
gfCNCPoint3[28361] = {X 390.4552, Y 8.2946, Z -4.6667, A 0.000, B 0.000, C 0.000 }
gfCNCPoint3[28362] = {X 391.3683, Y 7.9751, Z -4.6667, A 0.000, B 0.000, C 0.000 }
gfCNCPoint3[28363] = {X 392.3296, Y 7.8668, Z -4.6667, A 0.000, B 0.000, C 0.000 }
gfCNCPoint3[28364] = {X 399.1118, Y 7.8668, Z -4.6667, A 0.000, B 0.000, C 0.000 }
gfCNCPoint3[28365] = {X 400.0730, Y 7.9751, Z -4.6667, A 0.000, B 0.000, C 0.000 }
gfCNCPoint3[28366] = {X 400.9861, Y 8.2946, Z -4.6667, A 0.000, B 0.000, C 0.000 }
gfCNCPoint3[28367] = {X 401.8052, Y 8.8093, Z -4.6667, A 0.000, B 0.000, C 0.000 }
gfCNCPoint3[28368] = {X 402.4893, Y 9.4933, Z -4.6667, A 0.000, B 0.000, C 0.000 }
gfCNCPoint3[28369] = {X 403.0039, Y 10.3124, Z -4.6667, A 0.000, B 0.000, C 0.000 }
gfCNCPoint3[28370] = {X 403.3234, Y 11.2255, Z -4.6667, A 0.000, B 0.000, C 0.000 }
gfCNCPoint3[28371] = {X 403.4318, Y 12.1868, Z -4.6667, A 0.000, B 0.000, C 0.000 }
gfCNCPoint3[28372] = {X 403.4318, Y 12.9781, Z -4.6667, A 0.000, B 0.000, C 0.000 }
gfCNCPoint3[28373] = {X 403.3293, Y 13.9134, Z -4.6667, A 0.000, B 0.000, C 0.000 }
gfCNCPoint3[28374] = {X 403.0267, Y 14.8043, Z -4.6667, A 0.000, B 0.000, C 0.000 }
gfCNCPoint3[28375] = {X 405.3564, Y 18.8230, Z -4.6667, A 0.000, B 0.000, C 0.000 }
gfCNCPoint3[28376] = {X 407.8734, Y 14.7538, Z -4.6667, A 0.000, B 0.000, C 0.000 }
gfCNCPoint3[28377] = {X 407.5920, Y 13.9044, Z -4.6667, A 0.000, B 0.000, C 0.000 }
gfCNCPoint3[28378] = {X 407.4917, Y 13.0151, Z -4.6667, A 0.000, B 0.000, C 0.000 }
gfCNCPoint3[28379] = {X 407.4915, Y 12.1868, Z -4.6667, A 0.000, B 0.000, C 0.000 }
gfCNCPoint3[28380] = {X 407.5999, Y 11.2255, Z -4.6667, A 0.000, B 0.000, C 0.000 }
gfCNCPoint3[28381] = {X 407.9194, Y 10.3124, Z -4.6667, A 0.000, B 0.000, C 0.000 }
gfCNCPoint3[28382] = {X 408.4340, Y 9.4933, Z -4.6667, A 0.000, B 0.000, C 0.000 }
gfCNCPoint3[28383] = {X 409.1181, Y 8.8093, Z -4.6667, A 0.000, B 0.000, C 0.000 }
gfCNCPoint3[28384] = {X 409.9372, Y 8.2946, Z -4.6667, A 0.000, B 0.000, C 0.000 }
gfCNCPoint3[28385] = {X 410.8502, Y 7.9751, Z -4.6667, A 0.000, B 0.000, C 0.000 }
gfCNCPoint3[28386] = {X 411.8115, Y 7.8668, Z -4.6667, A 0.000, B 0.000, C 0.000 }
gfCNCPoint3[28387] = {X 419.3245, Y 7.8668, Z -4.6667, A 0.000, B 0.000, C 0.000 }
gfCNCPoint3[28388] = {X 420.2858, Y 7.9751, Z -4.6667, A 0.000, B 0.000, C 0.000 }
gfCNCPoint3[28389] = {X 421.1988, Y 8.2946, Z -4.6667, A 0.000, B 0.000, C 0.000 }
gfCNCPoint3[28390] = {X 422.0179, Y 8.8093, Z -4.6667, A 0.000, B 0.000, C 0.000 }
gfCNCPoint3[28391] = {X 422.7020, Y 9.4933, Z -4.6667, A 0.000, B 0.000, C 0.000 }
gfCNCPoint3[28392] = {X 423.2166, Y 10.3124, Z -4.6667, A 0.000, B 0.000, C 0.000 }
gfCNCPoint3[28393] = {X 423.5361, Y 11.2255, Z -4.6667, A 0.000, B 0.000, C 0.000 }
gfCNCPoint3[28394] = {X 423.6445, Y 12.1868, Z -4.6667, A 0.000, B 0.000, C 0.000 }
gfCNCPoint3[28395] = {X 423.6445, Y 12.9803, Z -4.6667, A 0.000, B 0.000, C 0.000 }
gfCNCPoint3[28396] = {X 423.5515, Y 13.8468, Z -4.6667, A 0.000, B 0.000, C 0.000 }
gfCNCPoint3[28397] = {X 423.2890, Y 14.6779, Z -4.6667, A 0.000, B 0.000, C 0.000 }
gfCNCPoint3[28398] = {X 422.8673, Y 15.4405, Z -4.6667, A 0.000, B 0.000, C 0.000 }
gfCNCPoint3[28399] = {X 422.3030, Y 16.1047, Z -4.6667, A 0.000, B 0.000, C 0.000 }
gfCNCPoint3[28400] = {X 421.6185, Y 16.6442, Z -4.6667, A 0.000, B 0.000, C 0.000 }
gfCNCPoint3[28401] = {X 420.8409, Y 17.0376, Z -4.6667, A 0.000, B 0.000, C 0.000 }
gfCNCPoint3[28402] = {X 420.1245, Y 18.0010, Z -4.6667, A 0.000, B 0.000, C 0.000 }
gfCNCPoint3[28403] = {X 419.4762, Y 19.0115, Z -4.6667, A 0.000, B 0.000, C 0.000 }
gfCNCPoint3[28404] = {X 417.9942, Y 21.4110, Z -4.6667, A 0.000, B 0.000, C 0.000 }
gfCNCPoint3[28405] = {X 416.1507, Y 24.3717, Z -4.6667, A 0.000, B 0.000, C 0.000 }
gfCNCPoint3[28406] = {X 419.5462, Y 26.4860, Z -4.6667, A 0.000, B 0.000, C 0.000 }
gfCNCPoint3[28407] = {X 416.0828, Y 24.3294, Z -4.6667, A 0.000, B 0.000, C 0.000 }
gfCNCPoint3[28408] = {X 411.4669, Y 31.7422, Z -4.6667, A 0.000, B 0.000, C 0.000 }
gfCNCPoint3[28409] = {X 411.4676, Y 40.9346, Z -4.6667, A 0.000, B 0.000, C 0.000 }
gfCNCPoint3[28410] = {X 412.1054, Y 41.6101, Z -4.6667, A 0.000, B 0.000, C 0.000 }
gfCNCPoint3[28411] = {X 412.5856, Y 42.4053, Z -4.6667, A 0.000, B 0.000, C 0.000 }
gfCNCPoint3[28412] = {X 412.8866, Y 43.2842, Z -4.6667, A 0.000, B 0.000, C 0.000 }
gfCNCPoint3[28413] = {X 412.9947, Y 44.2069, Z -4.6667, A 0.000, B 0.000, C 0.000 }
gfCNCPoint3[28414] = {X 412.9947, Y 45.0002, Z -4.6667, A 0.000, B 0.000, C 0.000 }
gfCNCPoint3[28415] = {X 412.8883, Y 45.9436, Z -4.6667, A 0.000, B 0.000, C 0.000 }
gfCNCPoint3[28416] = {X 412.5747, Y 46.8398, Z -4.6667, A 0.000, B 0.000, C 0.000 }
gfCNCPoint3[28417] = {X 412.0696, Y 47.6437, Z -4.6667, A 0.000, B 0.000, C 0.000 }
gfCNCPoint3[28418] = {X 411.3982, Y 48.3150, Z -4.6667, A 0.000, B 0.000, C 0.000 }
gfCNCPoint3[28419] = {X 410.5943, Y 48.8201, Z -4.6667, A 0.000, B 0.000, C 0.000 }
gfCNCPoint3[28420] = {X 409.6981, Y 49.1337, Z -4.6667, A 0.000, B 0.000, C 0.000 }
gfCNCPoint3[28421] = {X 408.7547, Y 49.2400, Z -4.6667, A 0.000, B 0.000, C 0.000 }
gfCNCPoint3[28422] = {X 402.3112, Y 49.2400, Z -4.6667, A 0.000, B 0.000, C 0.000 }
gfCNCPoint3[28423] = {X 401.3723, Y 49.1347, Z -4.6667, A 0.000, B 0.000, C 0.000 }
gfCNCPoint3[28424] = {X 400.4800, Y 48.8242, Z -4.6667, A 0.000, B 0.000, C 0.000 }
gfCNCPoint3[28425] = {X 399.6786, Y 48.3237, Z -4.6667, A 0.000, B 0.000, C 0.000 }
gfCNCPoint3[28426] = {X 399.0080, Y 47.6582, Z -4.6667, A 0.000, B 0.000, C 0.000 }
gfCNCPoint3[28427] = {X 398.5013, Y 46.8608, Z -4.6667, A 0.000, B 0.000, C 0.000 }
gfCNCPoint3[28428] = {X 398.1839, Y 45.9709, Z -4.6667, A 0.000, B 0.000, C 0.000 }
gfCNCPoint3[28429] = {X 398.0713, Y 45.0329, Z -4.6667, A 0.000, B 0.000, C 0.000 }
gfCNCPoint3[28430] = {X 398.0716, Y 44.1538, Z -4.6667, A 0.000, B 0.000, C 0.000 }
gfCNCPoint3[28431] = {X 398.1815, Y 43.2480, Z -4.6667, A 0.000, B 0.000, C 0.000 }
gfCNCPoint3[28432] = {X 398.4827, Y 42.3867, Z -4.6667, A 0.000, B 0.000, C 0.000 }
gfCNCPoint3[28433] = {X 398.9612, Y 41.6098, Z -4.6667, A 0.000, B 0.000, C 0.000 }
gfCNCPoint3[28434] = {X 399.5948, Y 40.9532, Z -4.6667, A 0.000, B 0.000, C 0.000 }
gfCNCPoint3[28435] = {X 399.5528, Y 31.5788, Z -4.6667, A 0.000, B 0.000, C 0.000 }
gfCNCPoint3[28436] = {X 393.5847, Y 21.2007, Z -4.6667, A 0.000, B 0.000, C 0.000 }
gfCNCPoint3[28437] = {X 392.6965, Y 19.6897, Z -4.6667, A 0.000, B 0.000, C 0.000 }
gfCNCPoint3[28438] = {X 391.7796, Y 18.1959, Z -4.6667, A 0.000, B 0.000, C 0.000 }
gfCNCPoint3[28439] = {X 391.2871, Y 17.5121, Z -4.6667, A 0.000, B 0.000, C 0.000 }
gfCNCPoint3[28440] = {X 390.7112, Y 16.8970, Z -4.6667, A 0.000, B 0.000, C 0.000 }
gfCNCPoint3[28441] = {X 389.8467, Y 16.4149, Z -4.6667, A 0.000, B 0.000, C 0.000 }
gfCNCPoint3[28442] = {X 389.1175, Y 15.7456, Z -4.6667, A 0.000, B 0.000, C 0.000 }
gfCNCPoint3[28443] = {X 388.5633, Y 14.9255, Z -4.6667, A 0.000, B 0.000, C 0.000 }
gfCNCPoint3[28444] = {X 388.2144, Y 13.9992, Z -4.6667, A 0.000, B 0.000, C 0.000 }
gfCNCPoint3[28445] = {X 388.0898, Y 13.0173, Z -4.6667, A 0.000, B 0.000, C 0.000 }
gfCNCPoint3[28446] = {X 388.0896, Y 12.1868, Z -4.6667, A 0.000, B 0.000, C 0.000 }
gfCNCPoint3[28447] = {X 388.1959, Y 11.2433, Z -4.6667, A 0.000, B 0.000, C 0.000 }
gfCNCPoint3[28448] = {X 388.5095, Y 10.3472, Z -4.6667, A 0.000, B 0.000, C 0.000 }
gfCNCPoint3[28449] = {X 389.0147, Y 9.5432, Z -4.6667, A 0.000, B 0.000, C 0.000 }
gfCNCPoint3[28450] = {X 389.6860, Y 8.8719, Z -4.6667, A 0.000, B 0.000, C 0.000 }
gfCNCPoint3[28451] = {X 390.4900, Y 8.3667, Z -4.6667, A 0.000, B 0.000, C 0.000 }
gfCNCPoint3[28452] = {X 391.3861, Y 8.0531, Z -4.6667, A 0.000, B 0.000, C 0.000 }
gfCNCPoint3[28453] = {X 392.3296, Y 7.9468, Z -4.6667, A 0.000, B 0.000, C 0.000 }
gfCNCPoint3[28454] = {X 399.1118, Y 7.9468, Z -4.6667, A 0.000, B 0.000, C 0.000 }
gfCNCPoint3[28455] = {X 400.0552, Y 8.0531, Z -4.6667, A 0.000, B 0.000, C 0.000 }
gfCNCPoint3[28456] = {X 400.9514, Y 8.3667, Z -4.6667, A 0.000, B 0.000, C 0.000 }
gfCNCPoint3[28457] = {X 401.7554, Y 8.8718, Z -4.6667, A 0.000, B 0.000, C 0.000 }
gfCNCPoint3[28458] = {X 402.4267, Y 9.5432, Z -4.6667, A 0.000, B 0.000, C 0.000 }
gfCNCPoint3[28459] = {X 402.9319, Y 10.3471, Z -4.6667, A 0.000, B 0.000, C 0.000 }
gfCNCPoint3[28460] = {X 403.2455, Y 11.2433, Z -4.6667, A 0.000, B 0.000, C 0.000 }
gfCNCPoint3[28461] = {X 403.3518, Y 12.1868, Z -4.6667, A 0.000, B 0.000, C 0.000 }
gfCNCPoint3[28462] = {X 403.3518, Y 12.9781, Z -4.6667, A 0.000, B 0.000, C 0.000 }
gfCNCPoint3[28463] = {X 403.2466, Y 13.9164, Z -4.6667, A 0.000, B 0.000, C 0.000 }
gfCNCPoint3[28464] = {X 402.9365, Y 14.8081, Z -4.6667, A 0.000, B 0.000, C 0.000 }
gfCNCPoint3[28465] = {X 405.3541, Y 18.9787, Z -4.6667, A 0.000, B 0.000, C 0.000 }
gfCNCPoint3[28466] = {X 407.9640, Y 14.7595, Z -4.6667, A 0.000, B 0.000, C 0.000 }
gfCNCPoint3[28467] = {X 407.6748, Y 13.9079, Z -4.6667, A 0.000, B 0.000, C 0.000 }
gfCNCPoint3[28468] = {X 407.5717, Y 13.0144, Z -4.6667, A 0.000, B 0.000, C 0.000 }
gfCNCPoint3[28469] = {X 407.5715, Y 12.1868, Z -4.6667, A 0.000, B 0.000, C 0.000 }
gfCNCPoint3[28470] = {X 407.6778, Y 11.2433, Z -4.6667, A 0.000, B 0.000, C 0.000 }
gfCNCPoint3[28471] = {X 407.9914, Y 10.3471, Z -4.6667, A 0.000, B 0.000, C 0.000 }
gfCNCPoint3[28472] = {X 408.4966, Y 9.5432, Z -4.6667, A 0.000, B 0.000, C 0.000 }
gfCNCPoint3[28473] = {X 409.1679, Y 8.8718, Z -4.6667, A 0.000, B 0.000, C 0.000 }
gfCNCPoint3[28474] = {X 409.9719, Y 8.3667, Z -4.6667, A 0.000, B 0.000, C 0.000 }
gfCNCPoint3[28475] = {X 410.8681, Y 8.0531, Z -4.6667, A 0.000, B 0.000, C 0.000 }
gfCNCPoint3[28476] = {X 411.8115, Y 7.9468, Z -4.6667, A 0.000, B 0.000, C 0.000 }
gfCNCPoint3[28477] = {X 419.3245, Y 7.9468, Z -4.6667, A 0.000, B 0.000, C 0.000 }
gfCNCPoint3[28478] = {X 420.2679, Y 8.0531, Z -4.6667, A 0.000, B 0.000, C 0.000 }
gfCNCPoint3[28479] = {X 421.1641, Y 8.3667, Z -4.6667, A 0.000, B 0.000, C 0.000 }
gfCNCPoint3[28480] = {X 421.9681, Y 8.8718, Z -4.6667, A 0.000, B 0.000, C 0.000 }
gfCNCPoint3[28481] = {X 422.6394, Y 9.5432, Z -4.6667, A 0.000, B 0.000, C 0.000 }
gfCNCPoint3[28482] = {X 423.1446, Y 10.3471, Z -4.6667, A 0.000, B 0.000, C 0.000 }
gfCNCPoint3[28483] = {X 423.4582, Y 11.2433, Z -4.6667, A 0.000, B 0.000, C 0.000 }
gfCNCPoint3[28484] = {X 423.5645, Y 12.1868, Z -4.6667, A 0.000, B 0.000, C 0.000 }
gfCNCPoint3[28485] = {X 423.5645, Y 12.9797, Z -4.6667, A 0.000, B 0.000, C 0.000 }
gfCNCPoint3[28486] = {X 423.4725, Y 13.8339, Z -4.6667, A 0.000, B 0.000, C 0.000 }
gfCNCPoint3[28487] = {X 423.2127, Y 14.6529, Z -4.6667, A 0.000, B 0.000, C 0.000 }
gfCNCPoint3[28488] = {X 422.7953, Y 15.4039, Z -4.6667, A 0.000, B 0.000, C 0.000 }
gfCNCPoint3[28489] = {X 422.2372, Y 16.0571, Z -4.6667, A 0.000, B 0.000, C 0.000 }
gfCNCPoint3[28490] = {X 421.5604, Y 16.5863, Z -4.6667, A 0.000, B 0.000, C 0.000 }
gfCNCPoint3[28491] = {X 420.7920, Y 16.9706, Z -4.6667, A 0.000, B 0.000, C 0.000 }
gfCNCPoint3[28492] = {X 420.0651, Y 17.9463, Z -4.6667, A 0.000, B 0.000, C 0.000 }
gfCNCPoint3[28493] = {X 419.4078, Y 18.9700, Z -4.6667, A 0.000, B 0.000, C 0.000 }
gfCNCPoint3[28494] = {X 417.9262, Y 21.3689, Z -4.6667, A 0.000, B 0.000, C 0.000 }
gfCNCPoint3[28495] = {X 416.0828, Y 24.3294, Z -4.6667, A 0.000, B 0.000, C 0.000 }
gfCNCPoint3[28496] = {X 419.4783, Y 26.4437, Z -4.6667, A 0.000, B 0.000, C 0.000 }
gfCNCPoint3[28497] = {X 416.0149, Y 24.2871, Z -4.6667, A 0.000, B 0.000, C 0.000 }
gfCNCPoint3[28498] = {X 411.3869, Y 31.7194, Z -4.6667, A 0.000, B 0.000, C 0.000 }
gfCNCPoint3[28499] = {X 411.3876, Y 40.9717, Z -4.6667, A 0.000, B 0.000, C 0.000 }
gfCNCPoint3[28500] = {X 412.0249, Y 41.6367, Z -4.6667, A 0.000, B 0.000, C 0.000 }
gfCNCPoint3[28501] = {X 412.5053, Y 42.4225, Z -4.6667, A 0.000, B 0.000, C 0.000 }
gfCNCPoint3[28502] = {X 412.8066, Y 43.2930, Z -4.6667, A 0.000, B 0.000, C 0.000 }
gfCNCPoint3[28503] = {X 412.9147, Y 44.2077, Z -4.6667, A 0.000, B 0.000, C 0.000 }
gfCNCPoint3[28504] = {X 412.9147, Y 45.0002, Z -4.6667, A 0.000, B 0.000, C 0.000 }
gfCNCPoint3[28505] = {X 412.8103, Y 45.9258, Z -4.6667, A 0.000, B 0.000, C 0.000 }
gfCNCPoint3[28506] = {X 412.5027, Y 46.8051, Z -4.6667, A 0.000, B 0.000, C 0.000 }
gfCNCPoint3[28507] = {X 412.0070, Y 47.5938, Z -4.6667, A 0.000, B 0.000, C 0.000 }
gfCNCPoint3[28508] = {X 411.3483, Y 48.2525, Z -4.6667, A 0.000, B 0.000, C 0.000 }
gfCNCPoint3[28509] = {X 410.5596, Y 48.7480, Z -4.6667, A 0.000, B 0.000, C 0.000 }
gfCNCPoint3[28510] = {X 409.6803, Y 49.0557, Z -4.6667, A 0.000, B 0.000, C 0.000 }
gfCNCPoint3[28511] = {X 408.7547, Y 49.1600, Z -4.6667, A 0.000, B 0.000, C 0.000 }
gfCNCPoint3[28512] = {X 402.3112, Y 49.1600, Z -4.6667, A 0.000, B 0.000, C 0.000 }
gfCNCPoint3[28513] = {X 401.3900, Y 49.0567, Z -4.6667, A 0.000, B 0.000, C 0.000 }
gfCNCPoint3[28514] = {X 400.5146, Y 48.7520, Z -4.6667, A 0.000, B 0.000, C 0.000 }
gfCNCPoint3[28515] = {X 399.7283, Y 48.2610, Z -4.6667, A 0.000, B 0.000, C 0.000 }
gfCNCPoint3[28516] = {X 399.0703, Y 47.6081, Z -4.6667, A 0.000, B 0.000, C 0.000 }
gfCNCPoint3[28517] = {X 398.5732, Y 46.8257, Z -4.6667, A 0.000, B 0.000, C 0.000 }
gfCNCPoint3[28518] = {X 398.2617, Y 45.9526, Z -4.6667, A 0.000, B 0.000, C 0.000 }
gfCNCPoint3[28519] = {X 398.1513, Y 45.0322, Z -4.6667, A 0.000, B 0.000, C 0.000 }
gfCNCPoint3[28520] = {X 398.1516, Y 44.1549, Z -4.6667, A 0.000, B 0.000, C 0.000 }
gfCNCPoint3[28521] = {X 398.2616, Y 43.2570, Z -4.6667, A 0.000, B 0.000, C 0.000 }
gfCNCPoint3[28522] = {X 398.5630, Y 42.4041, Z -4.6667, A 0.000, B 0.000, C 0.000 }
gfCNCPoint3[28523] = {X 399.0417, Y 41.6366, Z -4.6667, A 0.000, B 0.000, C 0.000 }
gfCNCPoint3[28524] = {X 399.6750, Y 40.9907, Z -4.6667, A 0.000, B 0.000, C 0.000 }
gfCNCPoint3[28525] = {X 399.6327, Y 31.5573, Z -4.6667, A 0.000, B 0.000, C 0.000 }
gfCNCPoint3[28526] = {X 393.6541, Y 21.1608, Z -4.6667, A 0.000, B 0.000, C 0.000 }
gfCNCPoint3[28527] = {X 392.7651, Y 19.6485, Z -4.6667, A 0.000, B 0.000, C 0.000 }
gfCNCPoint3[28528] = {X 391.8474, Y 18.1534, Z -4.6667, A 0.000, B 0.000, C 0.000 }
gfCNCPoint3[28529] = {X 391.3442, Y 17.4556, Z -4.6667, A 0.000, B 0.000, C 0.000 }
gfCNCPoint3[28530] = {X 390.7551, Y 16.8286, Z -4.6667, A 0.000, B 0.000, C 0.000 }
gfCNCPoint3[28531] = {X 389.9030, Y 16.3569, Z -4.6667, A 0.000, B 0.000, C 0.000 }
gfCNCPoint3[28532] = {X 389.1838, Y 15.7000, Z -4.6667, A 0.000, B 0.000, C 0.000 }
gfCNCPoint3[28533] = {X 388.6371, Y 14.8939, Z -4.6667, A 0.000, B 0.000, C 0.000 }
gfCNCPoint3[28534] = {X 388.2928, Y 13.9828, Z -4.6667, A 0.000, B 0.000, C 0.000 }
gfCNCPoint3[28535] = {X 388.1698, Y 13.0166, Z -4.6667, A 0.000, B 0.000, C 0.000 }
gfCNCPoint3[28536] = {X 388.1696, Y 12.1868, Z -4.6667, A 0.000, B 0.000, C 0.000 }
gfCNCPoint3[28537] = {X 388.2739, Y 11.2611, Z -4.6667, A 0.000, B 0.000, C 0.000 }
gfCNCPoint3[28538] = {X 388.5816, Y 10.3819, Z -4.6667, A 0.000, B 0.000, C 0.000 }
gfCNCPoint3[28539] = {X 389.0772, Y 9.5931, Z -4.6667, A 0.000, B 0.000, C 0.000 }
gfCNCPoint3[28540] = {X 389.7359, Y 8.9344, Z -4.6667, A 0.000, B 0.000, C 0.000 }
gfCNCPoint3[28541] = {X 390.5247, Y 8.4388, Z -4.6667, A 0.000, B 0.000, C 0.000 }
gfCNCPoint3[28542] = {X 391.4039, Y 8.1311, Z -4.6667, A 0.000, B 0.000, C 0.000 }
gfCNCPoint3[28543] = {X 392.3296, Y 8.0268, Z -4.6667, A 0.000, B 0.000, C 0.000 }
gfCNCPoint3[28544] = {X 399.1118, Y 8.0268, Z -4.6667, A 0.000, B 0.000, C 0.000 }
gfCNCPoint3[28545] = {X 400.0374, Y 8.1311, Z -4.6667, A 0.000, B 0.000, C 0.000 }
gfCNCPoint3[28546] = {X 400.9167, Y 8.4388, Z -4.6667, A 0.000, B 0.000, C 0.000 }
gfCNCPoint3[28547] = {X 401.7055, Y 8.9344, Z -4.6667, A 0.000, B 0.000, C 0.000 }
gfCNCPoint3[28548] = {X 402.3642, Y 9.5931, Z -4.6667, A 0.000, B 0.000, C 0.000 }
gfCNCPoint3[28549] = {X 402.8598, Y 10.3819, Z -4.6667, A 0.000, B 0.000, C 0.000 }
gfCNCPoint3[28550] = {X 403.1675, Y 11.2611, Z -4.6667, A 0.000, B 0.000, C 0.000 }
gfCNCPoint3[28551] = {X 403.2718, Y 12.1868, Z -4.6667, A 0.000, B 0.000, C 0.000 }
gfCNCPoint3[28552] = {X 403.2718, Y 12.9781, Z -4.6667, A 0.000, B 0.000, C 0.000 }
gfCNCPoint3[28553] = {X 403.1639, Y 13.9192, Z -4.6667, A 0.000, B 0.000, C 0.000 }
gfCNCPoint3[28554] = {X 402.8459, Y 14.8115, Z -4.6667, A 0.000, B 0.000, C 0.000 }
gfCNCPoint3[28555] = {X 405.3519, Y 19.1344, Z -4.6667, A 0.000, B 0.000, C 0.000 }
gfCNCPoint3[28556] = {X 408.0548, Y 14.7648, Z -4.6667, A 0.000, B 0.000, C 0.000 }
gfCNCPoint3[28557] = {X 407.7576, Y 13.9113, Z -4.6667, A 0.000, B 0.000, C 0.000 }
gfCNCPoint3[28558] = {X 407.6517, Y 13.0137, Z -4.6667, A 0.000, B 0.000, C 0.000 }
gfCNCPoint3[28559] = {X 407.6515, Y 12.1868, Z -4.6667, A 0.000, B 0.000, C 0.000 }
gfCNCPoint3[28560] = {X 407.7558, Y 11.2611, Z -4.6667, A 0.000, B 0.000, C 0.000 }
gfCNCPoint3[28561] = {X 408.0635, Y 10.3819, Z -4.6667, A 0.000, B 0.000, C 0.000 }
gfCNCPoint3[28562] = {X 408.5591, Y 9.5931, Z -4.6667, A 0.000, B 0.000, C 0.000 }
gfCNCPoint3[28563] = {X 409.2178, Y 8.9344, Z -4.6667, A 0.000, B 0.000, C 0.000 }
gfCNCPoint3[28564] = {X 410.0066, Y 8.4388, Z -4.6667, A 0.000, B 0.000, C 0.000 }
gfCNCPoint3[28565] = {X 410.8859, Y 8.1311, Z -4.6667, A 0.000, B 0.000, C 0.000 }
gfCNCPoint3[28566] = {X 411.8115, Y 8.0268, Z -4.6667, A 0.000, B 0.000, C 0.000 }
gfCNCPoint3[28567] = {X 419.3245, Y 8.0268, Z -4.6667, A 0.000, B 0.000, C 0.000 }
gfCNCPoint3[28568] = {X 420.2501, Y 8.1311, Z -4.6667, A 0.000, B 0.000, C 0.000 }
gfCNCPoint3[28569] = {X 421.1294, Y 8.4388, Z -4.6667, A 0.000, B 0.000, C 0.000 }
gfCNCPoint3[28570] = {X 421.9182, Y 8.9344, Z -4.6667, A 0.000, B 0.000, C 0.000 }
gfCNCPoint3[28571] = {X 422.5769, Y 9.5931, Z -4.6667, A 0.000, B 0.000, C 0.000 }
gfCNCPoint3[28572] = {X 423.0725, Y 10.3819, Z -4.6667, A 0.000, B 0.000, C 0.000 }
gfCNCPoint3[28573] = {X 423.3802, Y 11.2611, Z -4.6667, A 0.000, B 0.000, C 0.000 }
gfCNCPoint3[28574] = {X 423.4845, Y 12.1868, Z -4.6667, A 0.000, B 0.000, C 0.000 }
gfCNCPoint3[28575] = {X 423.4845, Y 12.9791, Z -4.6667, A 0.000, B 0.000, C 0.000 }
gfCNCPoint3[28576] = {X 423.3934, Y 13.8210, Z -4.6667, A 0.000, B 0.000, C 0.000 }
gfCNCPoint3[28577] = {X 423.1363, Y 14.6278, Z -4.6667, A 0.000, B 0.000, C 0.000 }
gfCNCPoint3[28578] = {X 422.7234, Y 15.3672, Z -4.6667, A 0.000, B 0.000, C 0.000 }
gfCNCPoint3[28579] = {X 422.1714, Y 16.0093, Z -4.6667, A 0.000, B 0.000, C 0.000 }
gfCNCPoint3[28580] = {X 421.5024, Y 16.5283, Z -4.6667, A 0.000, B 0.000, C 0.000 }
gfCNCPoint3[28581] = {X 420.7432, Y 16.9035, Z -4.6667, A 0.000, B 0.000, C 0.000 }
gfCNCPoint3[28582] = {X 420.0057, Y 17.8914, Z -4.6667, A 0.000, B 0.000, C 0.000 }
gfCNCPoint3[28583] = {X 419.3394, Y 18.9286, Z -4.6667, A 0.000, B 0.000, C 0.000 }
gfCNCPoint3[28584] = {X 417.8583, Y 21.3267, Z -4.6667, A 0.000, B 0.000, C 0.000 }
gfCNCPoint3[28585] = {X 416.0149, Y 24.2871, Z -4.6667, A 0.000, B 0.000, C 0.000 }
gfCNCPoint3[28586] = {X 419.4104, Y 26.4014, Z -4.6667, A 0.000, B 0.000, C 0.000 }
gfCNCPoint3[28587] = {X 415.9470, Y 24.2448, Z -4.6667, A 0.000, B 0.000, C 0.000 }
gfCNCPoint3[28588] = {X 411.3069, Y 31.6965, Z -4.6667, A 0.000, B 0.000, C 0.000 }
gfCNCPoint3[28589] = {X 411.3076, Y 41.0092, Z -4.6667, A 0.000, B 0.000, C 0.000 }
gfCNCPoint3[28590] = {X 411.9445, Y 41.6635, Z -4.6667, A 0.000, B 0.000, C 0.000 }
gfCNCPoint3[28591] = {X 412.4250, Y 42.4399, Z -4.6667, A 0.000, B 0.000, C 0.000 }
gfCNCPoint3[28592] = {X 412.7265, Y 43.3018, Z -4.6667, A 0.000, B 0.000, C 0.000 }
gfCNCPoint3[28593] = {X 412.8347, Y 44.2085, Z -4.6667, A 0.000, B 0.000, C 0.000 }
gfCNCPoint3[28594] = {X 412.8347, Y 45.0002, Z -4.6667, A 0.000, B 0.000, C 0.000 }
gfCNCPoint3[28595] = {X 412.7324, Y 45.9080, Z -4.6667, A 0.000, B 0.000, C 0.000 }
gfCNCPoint3[28596] = {X 412.4306, Y 46.7703, Z -4.6667, A 0.000, B 0.000, C 0.000 }
gfCNCPoint3[28597] = {X 411.9445, Y 47.5439, Z -4.6667, A 0.000, B 0.000, C 0.000 }
gfCNCPoint3[28598] = {X 411.2985, Y 48.1899, Z -4.6667, A 0.000, B 0.000, C 0.000 }
gfCNCPoint3[28599] = {X 410.5249, Y 48.6760, Z -4.6667, A 0.000, B 0.000, C 0.000 }
gfCNCPoint3[28600] = {X 409.6625, Y 48.9777, Z -4.6667, A 0.000, B 0.000, C 0.000 }
gfCNCPoint3[28601] = {X 408.7547, Y 49.0800, Z -4.6667, A 0.000, B 0.000, C 0.000 }
gfCNCPoint3[28602] = {X 402.3112, Y 49.0800, Z -4.6667, A 0.000, B 0.000, C 0.000 }
gfCNCPoint3[28603] = {X 401.4077, Y 48.9787, Z -4.6667, A 0.000, B 0.000, C 0.000 }
gfCNCPoint3[28604] = {X 400.5491, Y 48.6799, Z -4.6667, A 0.000, B 0.000, C 0.000 }
gfCNCPoint3[28605] = {X 399.7780, Y 48.1983, Z -4.6667, A 0.000, B 0.000, C 0.000 }
gfCNCPoint3[28606] = {X 399.1326, Y 47.5579, Z -4.6667, A 0.000, B 0.000, C 0.000 }
gfCNCPoint3[28607] = {X 398.6451, Y 46.7906, Z -4.6667, A 0.000, B 0.000, C 0.000 }
gfCNCPoint3[28608] = {X 398.3396, Y 45.9343, Z -4.6667, A 0.000, B 0.000, C 0.000 }
gfCNCPoint3[28609] = {X 398.2313, Y 45.0316, Z -4.6667, A 0.000, B 0.000, C 0.000 }
gfCNCPoint3[28610] = {X 398.2316, Y 44.1559, Z -4.6667, A 0.000, B 0.000, C 0.000 }
gfCNCPoint3[28611] = {X 398.3416, Y 43.2661, Z -4.6667, A 0.000, B 0.000, C 0.000 }
gfCNCPoint3[28612] = {X 398.6434, Y 42.4218, Z -4.6667, A 0.000, B 0.000, C 0.000 }
gfCNCPoint3[28613] = {X 399.1223, Y 41.6638, Z -4.6667, A 0.000, B 0.000, C 0.000 }
gfCNCPoint3[28614] = {X 399.7552, Y 41.0287, Z -4.6667, A 0.000, B 0.000, C 0.000 }
gfCNCPoint3[28615] = {X 399.7126, Y 31.5358, Z -4.6667, A 0.000, B 0.000, C 0.000 }
gfCNCPoint3[28616] = {X 393.7234, Y 21.1209, Z -4.6667, A 0.000, B 0.000, C 0.000 }
gfCNCPoint3[28617] = {X 392.8337, Y 19.6073, Z -4.6667, A 0.000, B 0.000, C 0.000 }
gfCNCPoint3[28618] = {X 391.9151, Y 18.1109, Z -4.6667, A 0.000, B 0.000, C 0.000 }
gfCNCPoint3[28619] = {X 391.4012, Y 17.3990, Z -4.6667, A 0.000, B 0.000, C 0.000 }
gfCNCPoint3[28620] = {X 390.7990, Y 16.7600, Z -4.6667, A 0.000, B 0.000, C 0.000 }
gfCNCPoint3[28621] = {X 389.9591, Y 16.2987, Z -4.6667, A 0.000, B 0.000, C 0.000 }
gfCNCPoint3[28622] = {X 389.2500, Y 15.6543, Z -4.6667, A 0.000, B 0.000, C 0.000 }
gfCNCPoint3[28623] = {X 388.7108, Y 14.8623, Z -4.6667, A 0.000, B 0.000, C 0.000 }
gfCNCPoint3[28624] = {X 388.3711, Y 13.9663, Z -4.6667, A 0.000, B 0.000, C 0.000 }
gfCNCPoint3[28625] = {X 388.2498, Y 13.0158, Z -4.6667, A 0.000, B 0.000, C 0.000 }
gfCNCPoint3[28626] = {X 388.2496, Y 12.1868, Z -4.6667, A 0.000, B 0.000, C 0.000 }
gfCNCPoint3[28627] = {X 388.3519, Y 11.2789, Z -4.6667, A 0.000, B 0.000, C 0.000 }
gfCNCPoint3[28628] = {X 388.6537, Y 10.4166, Z -4.6667, A 0.000, B 0.000, C 0.000 }
gfCNCPoint3[28629] = {X 389.1398, Y 9.6430, Z -4.6667, A 0.000, B 0.000, C 0.000 }
gfCNCPoint3[28630] = {X 389.7858, Y 8.9969, Z -4.6667, A 0.000, B 0.000, C 0.000 }
gfCNCPoint3[28631] = {X 390.5594, Y 8.5109, Z -4.6667, A 0.000, B 0.000, C 0.000 }
gfCNCPoint3[28632] = {X 391.4217, Y 8.2091, Z -4.6667, A 0.000, B 0.000, C 0.000 }
gfCNCPoint3[28633] = {X 392.3296, Y 8.1068, Z -4.6667, A 0.000, B 0.000, C 0.000 }
gfCNCPoint3[28634] = {X 399.1118, Y 8.1068, Z -4.6667, A 0.000, B 0.000, C 0.000 }
gfCNCPoint3[28635] = {X 400.0196, Y 8.2091, Z -4.6667, A 0.000, B 0.000, C 0.000 }
gfCNCPoint3[28636] = {X 400.8820, Y 8.5109, Z -4.6667, A 0.000, B 0.000, C 0.000 }
gfCNCPoint3[28637] = {X 401.6556, Y 8.9969, Z -4.6667, A 0.000, B 0.000, C 0.000 }
gfCNCPoint3[28638] = {X 402.3016, Y 9.6430, Z -4.6667, A 0.000, B 0.000, C 0.000 }
gfCNCPoint3[28639] = {X 402.7877, Y 10.4166, Z -4.6667, A 0.000, B 0.000, C 0.000 }
gfCNCPoint3[28640] = {X 403.0895, Y 11.2789, Z -4.6667, A 0.000, B 0.000, C 0.000 }
gfCNCPoint3[28641] = {X 403.1918, Y 12.1868, Z -4.6667, A 0.000, B 0.000, C 0.000 }
gfCNCPoint3[28642] = {X 403.1918, Y 12.9781, Z -4.6667, A 0.000, B 0.000, C 0.000 }
gfCNCPoint3[28643] = {X 403.0811, Y 13.9219, Z -4.6667, A 0.000, B 0.000, C 0.000 }
gfCNCPoint3[28644] = {X 402.7551, Y 14.8144, Z -4.6667, A 0.000, B 0.000, C 0.000 }
gfCNCPoint3[28645] = {X 405.3497, Y 19.2901, Z -4.6667, A 0.000, B 0.000, C 0.000 }
gfCNCPoint3[28646] = {X 408.1459, Y 14.7695, Z -4.6667, A 0.000, B 0.000, C 0.000 }
gfCNCPoint3[28647] = {X 408.1092, Y 14.6924, Z -4.6667, A 0.000, B 0.000, C 0.000 }
gfCNCPoint3[28648] = {X 408.0741, Y 14.6144, Z -4.6667, A 0.000, B 0.000, C 0.000 }
gfCNCPoint3[28649] = {X 407.8217, Y 13.8311, Z -4.6667, A 0.000, B 0.000, C 0.000 }
gfCNCPoint3[28650] = {X 407.7317, Y 13.0131, Z -4.6667, A 0.000, B 0.000, C 0.000 }
gfCNCPoint3[28651] = {X 407.7315, Y 12.1868, Z -4.6667, A 0.000, B 0.000, C 0.000 }
gfCNCPoint3[28652] = {X 407.8338, Y 11.2789, Z -4.6667, A 0.000, B 0.000, C 0.000 }
gfCNCPoint3[28653] = {X 408.1356, Y 10.4166, Z -4.6667, A 0.000, B 0.000, C 0.000 }
gfCNCPoint3[28654] = {X 408.6217, Y 9.6430, Z -4.6667, A 0.000, B 0.000, C 0.000 }
gfCNCPoint3[28655] = {X 409.2677, Y 8.9969, Z -4.6667, A 0.000, B 0.000, C 0.000 }
gfCNCPoint3[28656] = {X 410.0413, Y 8.5109, Z -4.6667, A 0.000, B 0.000, C 0.000 }
gfCNCPoint3[28657] = {X 410.9037, Y 8.2091, Z -4.6667, A 0.000, B 0.000, C 0.000 }
gfCNCPoint3[28658] = {X 411.8115, Y 8.1068, Z -4.6667, A 0.000, B 0.000, C 0.000 }
gfCNCPoint3[28659] = {X 419.3245, Y 8.1068, Z -4.6667, A 0.000, B 0.000, C 0.000 }
gfCNCPoint3[28660] = {X 420.2323, Y 8.2091, Z -4.6667, A 0.000, B 0.000, C 0.000 }
gfCNCPoint3[28661] = {X 421.0947, Y 8.5109, Z -4.6667, A 0.000, B 0.000, C 0.000 }
gfCNCPoint3[28662] = {X 421.8683, Y 8.9969, Z -4.6667, A 0.000, B 0.000, C 0.000 }
gfCNCPoint3[28663] = {X 422.5143, Y 9.6430, Z -4.6667, A 0.000, B 0.000, C 0.000 }
gfCNCPoint3[28664] = {X 423.0004, Y 10.4166, Z -4.6667, A 0.000, B 0.000, C 0.000 }
gfCNCPoint3[28665] = {X 423.3022, Y 11.2789, Z -4.6667, A 0.000, B 0.000, C 0.000 }
gfCNCPoint3[28666] = {X 423.4045, Y 12.1868, Z -4.6667, A 0.000, B 0.000, C 0.000 }
gfCNCPoint3[28667] = {X 423.4045, Y 12.9785, Z -4.6667, A 0.000, B 0.000, C 0.000 }
gfCNCPoint3[28668] = {X 423.3144, Y 13.8081, Z -4.6667, A 0.000, B 0.000, C 0.000 }
gfCNCPoint3[28669] = {X 423.0600, Y 14.6027, Z -4.6667, A 0.000, B 0.000, C 0.000 }
gfCNCPoint3[28670] = {X 422.6516, Y 15.3303, Z -4.6667, A 0.000, B 0.000, C 0.000 }
gfCNCPoint3[28671] = {X 422.1057, Y 15.9613, Z -4.6667, A 0.000, B 0.000, C 0.000 }
gfCNCPoint3[28672] = {X 421.4445, Y 16.4702, Z -4.6667, A 0.000, B 0.000, C 0.000 }
gfCNCPoint3[28673] = {X 420.6947, Y 16.8362, Z -4.6667, A 0.000, B 0.000, C 0.000 }
gfCNCPoint3[28674] = {X 419.9465, Y 17.8365, Z -4.6667, A 0.000, B 0.000, C 0.000 }
gfCNCPoint3[28675] = {X 419.2709, Y 18.8871, Z -4.6667, A 0.000, B 0.000, C 0.000 }
gfCNCPoint3[28676] = {X 417.7903, Y 21.2845, Z -4.6667, A 0.000, B 0.000, C 0.000 }
gfCNCPoint3[28677] = {X 415.9470, Y 24.2448, Z -4.6667, A 0.000, B 0.000, C 0.000 }
gfCNCPoint3[28678] = {X 419.3425, Y 26.3591, Z -4.6667, A 0.000, B 0.000, C 0.000 }
gfCNCPoint3[28679] = {X 415.8790, Y 24.2025, Z -4.6667, A 0.000, B 0.000, C 0.000 }
gfCNCPoint3[28680] = {X 411.2269, Y 31.6736, Z -4.6667, A 0.000, B 0.000, C 0.000 }
gfCNCPoint3[28681] = {X 411.2276, Y 41.0471, Z -4.6667, A 0.000, B 0.000, C 0.000 }
gfCNCPoint3[28682] = {X 411.8640, Y 41.6905, Z -4.6667, A 0.000, B 0.000, C 0.000 }
gfCNCPoint3[28683] = {X 412.3446, Y 42.4573, Z -4.6667, A 0.000, B 0.000, C 0.000 }
gfCNCPoint3[28684] = {X 412.6464, Y 43.3104, Z -4.6667, A 0.000, B 0.000, C 0.000 }
gfCNCPoint3[28685] = {X 412.7547, Y 44.2089, Z -4.6667, A 0.000, B 0.000, C 0.000 }
gfCNCPoint3[28686] = {X 412.7545, Y 45.0384, Z -4.6667, A 0.000, B 0.000, C 0.000 }
gfCNCPoint3[28687] = {X 412.6469, Y 45.9222, Z -4.6667, A 0.000, B 0.000, C 0.000 }
gfCNCPoint3[28688] = {X 412.3466, Y 46.7602, Z -4.6667, A 0.000, B 0.000, C 0.000 }
gfCNCPoint3[28689] = {X 411.8683, Y 47.5111, Z -4.6667, A 0.000, B 0.000, C 0.000 }
gfCNCPoint3[28690] = {X 411.2357, Y 48.1376, Z -4.6667, A 0.000, B 0.000, C 0.000 }
gfCNCPoint3[28691] = {X 410.4803, Y 48.6086, Z -4.6667, A 0.000, B 0.000, C 0.000 }
gfCNCPoint3[28692] = {X 409.6394, Y 48.9009, Z -4.6667, A 0.000, B 0.000, C 0.000 }
gfCNCPoint3[28693] = {X 408.7547, Y 49.0000, Z -4.6667, A 0.000, B 0.000, C 0.000 }
gfCNCPoint3[28694] = {X 402.3112, Y 49.0000, Z -4.6667, A 0.000, B 0.000, C 0.000 }
gfCNCPoint3[28695] = {X 401.4211, Y 48.8997, Z -4.6667, A 0.000, B 0.000, C 0.000 }
gfCNCPoint3[28696] = {X 400.5757, Y 48.6039, Z -4.6667, A 0.000, B 0.000, C 0.000 }
gfCNCPoint3[28697] = {X 399.8172, Y 48.1273, Z -4.6667, A 0.000, B 0.000, C 0.000 }
gfCNCPoint3[28698] = {X 399.1839, Y 47.4939, Z -4.6667, A 0.000, B 0.000, C 0.000 }
gfCNCPoint3[28699] = {X 398.7073, Y 46.7355, Z -4.6667, A 0.000, B 0.000, C 0.000 }
gfCNCPoint3[28700] = {X 398.4115, Y 45.8901, Z -4.6667, A 0.000, B 0.000, C 0.000 }
gfCNCPoint3[28701] = {X 398.3112, Y 45.0000, Z -4.6667, A 0.000, B 0.000, C 0.000 }
gfCNCPoint3[28702] = {X 398.3115, Y 44.1569, Z -4.6667, A 0.000, B 0.000, C 0.000 }
gfCNCPoint3[28703] = {X 398.4217, Y 43.2753, Z -4.6667, A 0.000, B 0.000, C 0.000 }
gfCNCPoint3[28704] = {X 398.7237, Y 42.4397, Z -4.6667, A 0.000, B 0.000, C 0.000 }
gfCNCPoint3[28705] = {X 399.2028, Y 41.6913, Z -4.6667, A 0.000, B 0.000, C 0.000 }
gfCNCPoint3[28706] = {X 399.8352, Y 41.0672, Z -4.6667, A 0.000, B 0.000, C 0.000 }
gfCNCPoint3[28707] = {X 399.8373, Y 31.5922, Z -4.6667, A 0.000, B 0.000, C 0.000 }
gfCNCPoint3[28708] = {X 393.7928, Y 21.0810, Z -4.6667, A 0.000, B 0.000, C 0.000 }
gfCNCPoint3[28709] = {X 392.9022, Y 19.5661, Z -4.6667, A 0.000, B 0.000, C 0.000 }
gfCNCPoint3[28710] = {X 391.9829, Y 18.0684, Z -4.6667, A 0.000, B 0.000, C 0.000 }
gfCNCPoint3[28711] = {X 391.4581, Y 17.3423, Z -4.6667, A 0.000, B 0.000, C 0.000 }
gfCNCPoint3[28712] = {X 390.8426, Y 16.6913, Z -4.6667, A 0.000, B 0.000, C 0.000 }
gfCNCPoint3[28713] = {X 390.0091, Y 16.2361, Z -4.6667, A 0.000, B 0.000, C 0.000 }
gfCNCPoint3[28714] = {X 389.3064, Y 15.5972, Z -4.6667, A 0.000, B 0.000, C 0.000 }
gfCNCPoint3[28715] = {X 388.7742, Y 14.8107, Z -4.6667, A 0.000, B 0.000, C 0.000 }
gfCNCPoint3[28716] = {X 388.4423, Y 13.9209, Z -4.6667, A 0.000, B 0.000, C 0.000 }
gfCNCPoint3[28717] = {X 388.3296, Y 12.9779, Z -4.6667, A 0.000, B 0.000, C 0.000 }
gfCNCPoint3[28718] = {X 388.3296, Y 12.1868, Z -4.6667, A 0.000, B 0.000, C 0.000 }
gfCNCPoint3[28719] = {X 388.4299, Y 11.2967, Z -4.6667, A 0.000, B 0.000, C 0.000 }
gfCNCPoint3[28720] = {X 388.7258, Y 10.4513, Z -4.6667, A 0.000, B 0.000, C 0.000 }
gfCNCPoint3[28721] = {X 389.2023, Y 9.6929, Z -4.6667, A 0.000, B 0.000, C 0.000 }
gfCNCPoint3[28722] = {X 389.8357, Y 9.0595, Z -4.6667, A 0.000, B 0.000, C 0.000 }
gfCNCPoint3[28723] = {X 390.5941, Y 8.5829, Z -4.6667, A 0.000, B 0.000, C 0.000 }
gfCNCPoint3[28724] = {X 391.4395, Y 8.2871, Z -4.6667, A 0.000, B 0.000, C 0.000 }
gfCNCPoint3[28725] = {X 392.3296, Y 8.1868, Z -4.6667, A 0.000, B 0.000, C 0.000 }
gfCNCPoint3[28726] = {X 399.1118, Y 8.1868, Z -4.6667, A 0.000, B 0.000, C 0.000 }
gfCNCPoint3[28727] = {X 400.0018, Y 8.2871, Z -4.6667, A 0.000, B 0.000, C 0.000 }
gfCNCPoint3[28728] = {X 400.8473, Y 8.5829, Z -4.6667, A 0.000, B 0.000, C 0.000 }
gfCNCPoint3[28729] = {X 401.6057, Y 9.0595, Z -4.6667, A 0.000, B 0.000, C 0.000 }
gfCNCPoint3[28730] = {X 402.2391, Y 9.6929, Z -4.6667, A 0.000, B 0.000, C 0.000 }
gfCNCPoint3[28731] = {X 402.7156, Y 10.4513, Z -4.6667, A 0.000, B 0.000, C 0.000 }
gfCNCPoint3[28732] = {X 403.0115, Y 11.2967, Z -4.6667, A 0.000, B 0.000, C 0.000 }
gfCNCPoint3[28733] = {X 403.1118, Y 12.1868, Z -4.6667, A 0.000, B 0.000, C 0.000 }
gfCNCPoint3[28734] = {X 403.1115, Y 13.0192, Z -4.6667, A 0.000, B 0.000, C 0.000 }
gfCNCPoint3[28735] = {X 402.9933, Y 13.9442, Z -4.6667, A 0.000, B 0.000, C 0.000 }
gfCNCPoint3[28736] = {X 402.6641, Y 14.8167, Z -4.6667, A 0.000, B 0.000, C 0.000 }
gfCNCPoint3[28737] = {X 405.2576, Y 19.3199, Z -4.6667, A 0.000, B 0.000, C 0.000 }
gfCNCPoint3[28738] = {X 405.3710, Y 19.4078, Z -4.6667, A 0.000, B 0.000, C 0.000 }
gfCNCPoint3[28739] = {X 408.1946, Y 14.8342, Z -4.6667, A 0.000, B 0.000, C 0.000 }
gfCNCPoint3[28740] = {X 408.2428, Y 14.7847, Z -4.6667, A 0.000, B 0.000, C 0.000 }
gfCNCPoint3[28741] = {X 408.1937, Y 14.6842, Z -4.6667, A 0.000, B 0.000, C 0.000 }
gfCNCPoint3[28742] = {X 408.1474, Y 14.5823, Z -4.6667, A 0.000, B 0.000, C 0.000 }
gfCNCPoint3[28743] = {X 407.8964, Y 13.7975, Z -4.6667, A 0.000, B 0.000, C 0.000 }
gfCNCPoint3[28744] = {X 407.8115, Y 12.9779, Z -4.6667, A 0.000, B 0.000, C 0.000 }
gfCNCPoint3[28745] = {X 407.8115, Y 12.1868, Z -4.6667, A 0.000, B 0.000, C 0.000 }
gfCNCPoint3[28746] = {X 407.9118, Y 11.2967, Z -4.6667, A 0.000, B 0.000, C 0.000 }
gfCNCPoint3[28747] = {X 408.2077, Y 10.4513, Z -4.6667, A 0.000, B 0.000, C 0.000 }
gfCNCPoint3[28748] = {X 408.6842, Y 9.6929, Z -4.6667, A 0.000, B 0.000, C 0.000 }
gfCNCPoint3[28749] = {X 409.3176, Y 9.0595, Z -4.6667, A 0.000, B 0.000, C 0.000 }
gfCNCPoint3[28750] = {X 410.0760, Y 8.5829, Z -4.6667, A 0.000, B 0.000, C 0.000 }
gfCNCPoint3[28751] = {X 410.9215, Y 8.2871, Z -4.6667, A 0.000, B 0.000, C 0.000 }
gfCNCPoint3[28752] = {X 411.8115, Y 8.1868, Z -4.6667, A 0.000, B 0.000, C 0.000 }
gfCNCPoint3[28753] = {X 419.3245, Y 8.1868, Z -4.6667, A 0.000, B 0.000, C 0.000 }
gfCNCPoint3[28754] = {X 420.2145, Y 8.2871, Z -4.6667, A 0.000, B 0.000, C 0.000 }
gfCNCPoint3[28755] = {X 421.0600, Y 8.5829, Z -4.6667, A 0.000, B 0.000, C 0.000 }
gfCNCPoint3[28756] = {X 421.8184, Y 9.0595, Z -4.6667, A 0.000, B 0.000, C 0.000 }
gfCNCPoint3[28757] = {X 422.4518, Y 9.6929, Z -4.6667, A 0.000, B 0.000, C 0.000 }
gfCNCPoint3[28758] = {X 422.9283, Y 10.4513, Z -4.6667, A 0.000, B 0.000, C 0.000 }
gfCNCPoint3[28759] = {X 423.2242, Y 11.2967, Z -4.6667, A 0.000, B 0.000, C 0.000 }
gfCNCPoint3[28760] = {X 423.3245, Y 12.1868, Z -4.6667, A 0.000, B 0.000, C 0.000 }
gfCNCPoint3[28761] = {X 423.3245, Y 12.9780, Z -4.6667, A 0.000, B 0.000, C 0.000 }
gfCNCPoint3[28762] = {X 423.1978, Y 13.9554, Z -4.6667, A 0.000, B 0.000, C 0.000 }
gfCNCPoint3[28763] = {X 422.8396, Y 14.8735, Z -4.6667, A 0.000, B 0.000, C 0.000 }
gfCNCPoint3[28764] = {X 422.2710, Y 15.6785, Z -4.6667, A 0.000, B 0.000, C 0.000 }
gfCNCPoint3[28765] = {X 421.5252, Y 16.3228, Z -4.6667, A 0.000, B 0.000, C 0.000 }
gfCNCPoint3[28766] = {X 420.6463, Y 16.7687, Z -4.6667, A 0.000, B 0.000, C 0.000 }
gfCNCPoint3[28767] = {X 419.8873, Y 17.7814, Z -4.6667, A 0.000, B 0.000, C 0.000 }
gfCNCPoint3[28768] = {X 419.2025, Y 18.8457, Z -4.6667, A 0.000, B 0.000, C 0.000 }
gfCNCPoint3[28769] = {X 417.7223, Y 21.2424, Z -4.6667, A 0.000, B 0.000, C 0.000 }
gfCNCPoint3[28770] = {X 415.8790, Y 24.2025, Z -4.6667, A 0.000, B 0.000, C 0.000 }
gfCNCPoint3[28771] = {X 419.3425, Y 26.3591, Z -4.6667, A 0.000, B 0.000, C 0.000 }
gfCNCPoint3[28772] = {X 419.3425, Y 26.3591, Z -1.6667, A 0.000, B 0.000, C 0.000 }
gfCNCPoint3[28773] = {X 419.3425, Y 26.3591, Z 11.0000, A 0.000, B 0.000, C 0.000 }
